LIN {X 0,Y 164.782,Z 136.258,A -85,B 0,C 180,E1 -23321.199,E2 -23321.199} C_VEL
LIN {X 0,Y 164.508,Z 136.296,A -85,B 0,C 180,E1 -23327.402,E2 -23327.402} C_VEL
LIN {X 0,Y 164.476,Z 136.307,A -85,B 0,C 180,E1 -23329.99,E2 -23329.99} C_VEL
LIN {X 0,Y 164.429,Z 136.475,A -85,B 0,C 180,E1 -23333.875,E2 -23333.875} C_VEL
LIN {X 0,Y 165.572,Z 139.373,A -85,B 0,C 180,E1 -23334.533,E2 -23334.533} C_VEL
LIN {X 0,Y 166.931,Z 141.256,A -85,B 0,C 180,E1 -23335.132,E2 -23335.132} C_VEL
LIN {X 0,Y 173.938,Z 153.479,A -85,B 0,C 180,E1 -23338.268,E2 -23338.268} C_VEL
LIN {X 0,Y 182.776,Z 169.655,A -85,B 0,C 180,E1 -23341.878,E2 -23341.878} C_VEL
LIN {X 0,Y 193.204,Z 190.491,A -85,B 0,C 180,E1 -23345.779,E2 -23345.779} C_VEL
LIN {X 0,Y 203.818,Z 212.836,A -85,B 0,C 180,E1 -23349.361,E2 -23349.361} C_VEL
LIN {X 0,Y 191.616,Z 314.791,A -85,B 0,C 180,E1 -23355.179,E2 -23355.179} C_VEL
LIN {X 0,Y 189.078,Z 333.623,A -85,B 0,C 180,E1 -23356.739,E2 -23356.739} C_VEL
LIN {X 0,Y 186.109,Z 350.938,A -85,B 0,C 180,E1 -23358.581,E2 -23358.581} C_VEL
LIN {X 0,Y 182.724,Z 368.577,A -85,B 0,C 180,E1 -23360.963,E2 -23360.963} C_VEL
LIN {X 0,Y 179.217,Z 384.609,A -85,B 0,C 180,E1 -23363.62,E2 -23363.62} C_VEL
LIN {X 0,Y 175.913,Z 399.098,A -85,B 0,C 180,E1 -23366.535,E2 -23366.535} C_VEL
LIN {X 0,Y 172.526,Z 413.606,A -85,B 0,C 180,E1 -23370.065,E2 -23370.065} C_VEL
LIN {X 0,Y 169.416,Z 427.579,A -85,B 0,C 180,E1 -23374.178,E2 -23374.178} C_VEL
LIN {X 0,Y 166.846,Z 439.432,A -85,B 0,C 180,E1 -23378.372,E2 -23378.372} C_VEL
LIN {X 0,Y 164.935,Z 449.571,A -85,B 0,C 180,E1 -23382.646,E2 -23382.646} C_VEL
LIN {X 0,Y 163.47,Z 459.455,A -85,B 0,C 180,E1 -23387.586,E2 -23387.586} C_VEL
LIN {X 0,Y 162.879,Z 465.778,A -85,B 0,C 180,E1 -23391.314,E2 -23391.314} C_VEL
LIN {X 0,Y 162.51,Z 472.942,A -85,B 0,C 180,E1 -23396.28,E2 -23396.28} C_VEL
LIN {X 0,Y 162.642,Z 478.87,A -85,B 0,C 180,E1 -23401.238,E2 -23401.238} C_VEL
LIN {X 0,Y 163.36,Z 483.627,A -85,B 0,C 180,E1 -23406.174,E2 -23406.174} C_VEL
LIN {X 0,Y 165.201,Z 488.286,A -85,B 0,C 180,E1 -23412.281,E2 -23412.281} C_VEL
LIN {X 0,Y 167.913,Z 491.025,A -85,B 0,C 180,E1 -23417.036,E2 -23417.036} C_VEL
LIN {X 0,Y 171.601,Z 493.04,A -85,B 0,C 180,E1 -23421.629,E2 -23421.629} C_VEL
LIN {X 0,Y 179.115,Z 494.623,A -85,B 0,C 180,E1 -23428.089,E2 -23428.089} C_VEL
LIN {X 0,Y 189.089,Z 494.613,A -85,B 0,C 180,E1 -23433.884,E2 -23433.884} C_VEL
LIN {X 0,Y 196.793,Z 493.837,A -85,B 0,C 180,E1 -23437.381,E2 -23437.381} C_VEL
LIN {X 0,Y 210.033,Z 491.428,A -85,B 0,C 180,E1 -23442.007,E2 -23442.007} C_VEL
LIN {X 0,Y 195.119,Z 497.326,A -85,B 0,C 180,E1 -23446.813,E2 -23446.813} C_VEL
LIN {X 0,Y 183.475,Z 501.617,A -85,B 0,C 180,E1 -23452.2,E2 -23452.2} C_VEL
LIN {X 0,Y 175.646,Z 504.236,A -85,B 0,C 180,E1 -23457.167,E2 -23457.167} C_VEL
LIN {X 0,Y 169.36,Z 505.964,A -85,B 0,C 180,E1 -23462.839,E2 -23462.839} C_VEL
LIN {X 0,Y 164.641,Z 506.692,A -85,B 0,C 180,E1 -23470.179,E2 -23470.179} C_VEL
LIN {X 0,Y 162.82,Z 505.777,A -85,B 0,C 180,E1 -23477.535,E2 -23477.535} C_VEL
LIN {X 0,Y 162.814,Z 504.732,A -85,B 0,C 180,E1 -23480.877,E2 -23480.877} C_VEL
LIN {X 0,Y 162.399,Z 503.811,A -85,B 0,C 180,E1 -23482.926,E2 -23482.926} C_VEL
LIN {X 0,Y 161.187,Z 502.51,A -85,B 0,C 180,E1 -23484.934,E2 -23484.934} C_VEL
LIN {X 0,Y 157.491,Z 497.688,A -85,B 0,C 180,E1 -23490.301,E2 -23490.301} C_VEL
LIN {X 0,Y 157.2,Z 496.337,A -85,B 0,C 180,E1 -23491.68,E2 -23491.68} C_VEL
LIN {X 0,Y 157.104,Z 492.695,A -85,B 0,C 180,E1 -23495.131,E2 -23495.131} C_VEL
LIN {X 0,Y 156.843,Z 485.87,A -85,B 0,C 180,E1 -23500.324,E2 -23500.324} C_VEL
LIN {X 0,Y 157.182,Z 479.569,A -85,B 0,C 180,E1 -23504.234,E2 -23504.234} C_VEL
LIN {X 0,Y 158.14,Z 470.979,A -85,B 0,C 180,E1 -23508.794,E2 -23508.794} C_VEL
LIN {X 0,Y 159.756,Z 460.712,A -85,B 0,C 180,E1 -23513.322,E2 -23513.322} C_VEL
LIN {X 0,Y 162.296,Z 448.632,A -85,B 0,C 180,E1 -23517.742,E2 -23517.742} C_VEL
LIN {X 0,Y 165.078,Z 436.661,A -85,B 0,C 180,E1 -23521.388,E2 -23521.388} C_VEL
LIN {X 0,Y 168.577,Z 422.487,A -85,B 0,C 180,E1 -23524.974,E2 -23524.974} C_VEL
LIN {X 0,Y 172.253,Z 407.32,A -85,B 0,C 180,E1 -23528.103,E2 -23528.103} C_VEL
LIN {X 0,Y 175.841,Z 391.722,A -85,B 0,C 180,E1 -23530.722,E2 -23530.722} C_VEL
LIN {X 0,Y 179.532,Z 374.404,A -85,B 0,C 180,E1 -23533.046,E2 -23533.046} C_VEL
LIN {X 0,Y 182.942,Z 356.554,A -85,B 0,C 180,E1 -23534.9,E2 -23534.9} C_VEL
LIN {X 0,Y 185.607,Z 338.247,A -85,B 0,C 180,E1 -23536.35,E2 -23536.35} C_VEL
LIN {X 0,Y 199.629,Z 227.884,A -85,B 0,C 180,E1 -23542.848,E2 -23542.848} C_VEL
LIN {X 0,Y 190.678,Z 205.57,A -85,B 0,C 180,E1 -23546.198,E2 -23546.198} C_VEL
LIN {X 0,Y 181.033,Z 183.19,A -85,B 0,C 180,E1 -23550.094,E2 -23550.094} C_VEL
LIN {X 0,Y 172.608,Z 164.737,A -85,B 0,C 180,E1 -23553.83,E2 -23553.83} C_VEL
LIN {X 0,Y 168.302,Z 156.399,A -85,B 0,C 180,E1 -23555.815,E2 -23555.815} C_VEL
LIN {X 0,Y 161.572,Z 145.068,A -85,B 0,C 180,E1 -23558.97,E2 -23558.97} C_VEL
LIN {X 0,Y 159.276,Z 141.104,A -85,B 0,C 180,E1 -23560.142,E2 -23560.142} C_VEL
LIN {X 0,Y 157.757,Z 138.666,A -85,B 0,C 180,E1 -23560.916,E2 -23560.916} C_VEL
LIN {X 0,Y 157.409,Z 137.193,A -85,B 0,C 180,E1 -23561.216,E2 -23561.216} C_VEL
LIN {X 0,Y 157.556,Z 137.159,A -85,B 0,C 180,E1 -23567.113,E2 -23567.113} C_VEL
LIN {X 0,Y 157.768,Z 137.14,A -85,B 0,C 180,E1 -23569.736,E2 -23569.736} C_VEL
LIN {X 0,Y 157.82,Z 137.138,A -85,B 0,C 180,E1 -23572.323,E2 -23572.323} C_VEL
LIN {X 0,Y 158.256,Z 137.083,A -85,B 0,C 180,E1 -23580,E2 -23580} C_VEL
LIN {X 0,Y 157.821,Z 137.137,A -85,B 0,C 180,E1 -23587.678,E2 -23587.678} C_VEL
LIN {X 0,Y 157.702,Z 137.147,A -85,B 0,C 180,E1 -23591.363,E2 -23591.363} C_VEL
LIN {X 0,Y 157.474,Z 137.18,A -85,B 0,C 180,E1 -23595.532,E2 -23595.532} C_VEL
LIN {X 0,Y 157.366,Z 137.196,A -85,B 0,C 180,E1 -23600.934,E2 -23600.934} C_VEL
LIN {X 0,Y 157.312,Z 137.2,A -85,B 0,C 180,E1 -23606.686,E2 -23606.686} C_VEL
LIN {X 0,Y 157.272,Z 137.2,A -85,B 0,C 180,E1 -23612.428,E2 -23612.428} C_VEL
LIN {X 0,Y 157.264,Z 137.206,A -85,B 0,C 180,E1 -23616.45,E2 -23616.45} C_VEL
LIN {X 0,Y 157.208,Z 137.214,A -85,B 0,C 180,E1 -23622.112,E2 -23622.112} C_VEL
LIN {X 0,Y 157.238,Z 137.205,A -85,B 0,C 180,E1 -23627.901,E2 -23627.901} C_VEL
LIN {X 0,Y 157.32,Z 137.189,A -85,B 0,C 180,E1 -23633.526,E2 -23633.526} C_VEL
LIN {X 0,Y 157.293,Z 137.204,A -85,B 0,C 180,E1 -23638.097,E2 -23638.097} C_VEL
LIN {X 0,Y 157.321,Z 137.198,A -85,B 0,C 180,E1 -23643.468,E2 -23643.468} C_VEL
LIN {X 0,Y 157.446,Z 137.178,A -85,B 0,C 180,E1 -23649.618,E2 -23649.618} C_VEL
LIN {X 0,Y 157.466,Z 137.175,A -85,B 0,C 180,E1 -23654.469,E2 -23654.469} C_VEL
LIN {X 0,Y 157.75,Z 137.146,A -85,B 0,C 180,E1 -23659.736,E2 -23659.736} C_VEL
LIN {X 0,Y 157.822,Z 137.133,A -85,B 0,C 180,E1 -23662.324,E2 -23662.324} C_VEL
LIN {X 0,Y 158.259,Z 137.083,A -85,B 0,C 180,E1 -23670.002,E2 -23670.002} C_VEL
LIN {X 0,Y 157.826,Z 137.141,A -85,B 0,C 180,E1 -23677.679,E2 -23677.679} C_VEL
LIN {X 0,Y 157.708,Z 137.139,A -85,B 0,C 180,E1 -23681.364,E2 -23681.364} C_VEL
LIN {X 0,Y 157.481,Z 137.184,A -85,B 0,C 180,E1 -23685.533,E2 -23685.533} C_VEL
LIN {X 0,Y 157.373,Z 137.195,A -85,B 0,C 180,E1 -23690.934,E2 -23690.934} C_VEL
LIN {X 0,Y 157.348,Z 137.194,A -85,B 0,C 180,E1 -23691.71,E2 -23691.71} C_VEL
LIN {X 0,Y 158.41,Z 140.134,A -85,B 0,C 180,E1 -23692.414,E2 -23692.414} C_VEL
LIN {X 0,Y 159.928,Z 142.172,A -85,B 0,C 180,E1 -23693.128,E2 -23693.128} C_VEL
LIN {X 0,Y 167.079,Z 154.486,A -85,B 0,C 180,E1 -23696.549,E2 -23696.549} C_VEL
LIN {X 0,Y 175.9,Z 170.567,A -85,B 0,C 180,E1 -23700.378,E2 -23700.378} C_VEL
LIN {X 0,Y 186.553,Z 191.815,A -85,B 0,C 180,E1 -23704.595,E2 -23704.595} C_VEL
LIN {X 0,Y 197.438,Z 214.94,A -85,B 0,C 180,E1 -23708.461,E2 -23708.461} C_VEL
LIN {X 0,Y 185.105,Z 314.275,A -85,B 0,C 180,E1 -23714.319,E2 -23714.319} C_VEL
LIN {X 0,Y 182.501,Z 333.276,A -85,B 0,C 180,E1 -23715.927,E2 -23715.927} C_VEL
LIN {X 0,Y 179.205,Z 352.05,A -85,B 0,C 180,E1 -23717.998,E2 -23717.998} C_VEL
LIN {X 0,Y 175.967,Z 368.444,A -85,B 0,C 180,E1 -23720.28,E2 -23720.28} C_VEL
LIN {X 0,Y 172.363,Z 384.5,A -85,B 0,C 180,E1 -23723.028,E2 -23723.028} C_VEL
LIN {X 0,Y 168.77,Z 399.805,A -85,B 0,C 180,E1 -23726.229,E2 -23726.229} C_VEL
LIN {X 0,Y 165.206,Z 414.682,A -85,B 0,C 180,E1 -23730.009,E2 -23730.009} C_VEL
LIN {X 0,Y 162.073,Z 428.527,A -85,B 0,C 180,E1 -23734.301,E2 -23734.301} C_VEL
LIN {X 0,Y 159.483,Z 440.457,A -85,B 0,C 180,E1 -23738.754,E2 -23738.754} C_VEL
LIN {X 0,Y 157.881,Z 449.027,A -85,B 0,C 180,E1 -23742.514,E2 -23742.514} C_VEL
LIN {X 0,Y 156.373,Z 459.064,A -85,B 0,C 180,E1 -23747.673,E2 -23747.673} C_VEL
LIN {X 0,Y 155.681,Z 466.451,A -85,B 0,C 180,E1 -23752.216,E2 -23752.216} C_VEL
LIN {X 0,Y 155.485,Z 473.586,A -85,B 0,C 180,E1 -23757.409,E2 -23757.409} C_VEL
LIN {X 0,Y 155.73,Z 479.475,A -85,B 0,C 180,E1 -23762.586,E2 -23762.586} C_VEL
LIN {X 0,Y 156.598,Z 484.232,A -85,B 0,C 180,E1 -23767.737,E2 -23767.737} C_VEL
LIN {X 0,Y 158.266,Z 488.082,A -85,B 0,C 180,E1 -23772.828,E2 -23772.828} C_VEL
LIN {X 0,Y 161.129,Z 491.113,A -85,B 0,C 180,E1 -23777.777,E2 -23777.777} C_VEL
LIN {X 0,Y 167.394,Z 494.193,A -85,B 0,C 180,E1 -23784.825,E2 -23784.825} C_VEL
LIN {X 0,Y 176.084,Z 495.685,A -85,B 0,C 180,E1 -23791.256,E2 -23791.256} C_VEL
LIN {X 0,Y 187.203,Z 495.638,A -85,B 0,C 180,E1 -23796.918,E2 -23796.918} C_VEL
LIN {X 0,Y 200.238,Z 494.178,A -85,B 0,C 180,E1 -23801.825,E2 -23801.825} C_VEL
LIN {X 0,Y 199.396,Z 494.527,A -85,B 0,C 180,E1 -23802.252,E2 -23802.252} C_VEL
LIN {X 0,Y 190.006,Z 497.729,A -85,B 0,C 180,E1 -23805.348,E2 -23805.348} C_VEL
LIN {X 0,Y 177.876,Z 501.623,A -85,B 0,C 180,E1 -23810.788,E2 -23810.788} C_VEL
LIN {X 0,Y 168.063,Z 504.222,A -85,B 0,C 180,E1 -23817.067,E2 -23817.067} C_VEL
LIN {X 0,Y 161.011,Z 505.535,A -85,B 0,C 180,E1 -23824.118,E2 -23824.118} C_VEL
LIN {X 0,Y 158.018,Z 505.611,A -85,B 0,C 180,E1 -23829.155,E2 -23829.155} C_VEL
LIN {X 0,Y 156.306,Z 505,A -85,B 0,C 180,E1 -23834.347,E2 -23834.347} C_VEL
LIN {X 0,Y 155.909,Z 503.121,A -85,B 0,C 180,E1 -23840.876,E2 -23840.876} C_VEL
LIN {X 0,Y 156.452,Z 501.308,A -85,B 0,C 180,E1 -23844.844,E2 -23844.844} C_VEL
LIN {X 0,Y 156.936,Z 499.805,A -85,B 0,C 180,E1 -23847.432,E2 -23847.432} C_VEL
LIN {X 0,Y 157.29,Z 497.859,A -85,B 0,C 180,E1 -23849.998,E2 -23849.998} C_VEL
LIN {X 0,Y 157.2,Z 496.337,A -85,B 0,C 180,E1 -23851.68,E2 -23851.68} C_VEL
LIN {X 0,Y 156.469,Z 494.187,A -85,B 0,C 180,E1 -23853.65,E2 -23853.65} C_VEL
LIN {X 0,Y 154.839,Z 491.662,A -85,B 0,C 180,E1 -23855.53,E2 -23855.53} C_VEL
LIN {X 0,Y 151.087,Z 485.896,A -85,B 0,C 180,E1 -23859.235,E2 -23859.235} C_VEL
LIN {X 0,Y 150.093,Z 482.788,A -85,B 0,C 180,E1 -23861.176,E2 -23861.176} C_VEL
LIN {X 0,Y 150.043,Z 481.776,A -85,B 0,C 180,E1 -23861.842,E2 -23861.842} C_VEL
LIN {X 0,Y 150.725,Z 473.135,A -85,B 0,C 180,E1 -23866.941,E2 -23866.941} C_VEL
LIN {X 0,Y 152.057,Z 463.428,A -85,B 0,C 180,E1 -23871.699,E2 -23871.699} C_VEL
LIN {X 0,Y 154.322,Z 452.034,A -85,B 0,C 180,E1 -23876.359,E2 -23876.359} C_VEL
LIN {X 0,Y 157.22,Z 439.664,A -85,B 0,C 180,E1 -23880.561,E2 -23880.561} C_VEL
LIN {X 0,Y 160.831,Z 425.013,A -85,B 0,C 180,E1 -23884.614,E2 -23884.614} C_VEL
LIN {X 0,Y 164.79,Z 408.962,A -85,B 0,C 180,E1 -23888.197,E2 -23888.197} C_VEL
LIN {X 0,Y 168.826,Z 392.119,A -85,B 0,C 180,E1 -23891.203,E2 -23891.203} C_VEL
LIN {X 0,Y 172.548,Z 375.19,A -85,B 0,C 180,E1 -23893.598,E2 -23893.598} C_VEL
LIN {X 0,Y 176.029,Z 357.565,A -85,B 0,C 180,E1 -23895.532,E2 -23895.532} C_VEL
LIN {X 0,Y 178.683,Z 340.392,A -85,B 0,C 180,E1 -23896.996,E2 -23896.996} C_VEL
LIN {X 0,Y 193.251,Z 229.764,A -85,B 0,C 180,E1 -23903.774,E2 -23903.774} C_VEL
LIN {X 0,Y 185.238,Z 209.471,A -85,B 0,C 180,E1 -23906.908,E2 -23906.908} C_VEL
LIN {X 0,Y 175.951,Z 187.639,A -85,B 0,C 180,E1 -23910.826,E2 -23910.826} C_VEL
LIN {X 0,Y 167.779,Z 169.366,A -85,B 0,C 180,E1 -23914.625,E2 -23914.625} C_VEL
LIN {X 0,Y 163.269,Z 160.612,A -85,B 0,C 180,E1 -23916.777,E2 -23916.777} C_VEL
LIN {X 0,Y 156.306,Z 148.806,A -85,B 0,C 180,E1 -23920.21,E2 -23920.21} C_VEL
LIN {X 0,Y 154.262,Z 145.429,A -85,B 0,C 180,E1 -23921.286,E2 -23921.286} C_VEL
LIN {X 0,Y 152.425,Z 142.211,A -85,B 0,C 180,E1 -23922.301,E2 -23922.301} C_VEL
LIN {X 0,Y 150.837,Z 139.865,A -85,B 0,C 180,E1 -23923.157,E2 -23923.157} C_VEL
LIN {X 0,Y 150.378,Z 138.061,A -85,B 0,C 180,E1 -23923.628,E2 -23923.628} C_VEL
LIN {X 0,Y 150.685,Z 138.018,A -85,B 0,C 180,E1 -23929.248,E2 -23929.248} C_VEL
LIN {X 0,Y 150.759,Z 138.019,A -85,B 0,C 180,E1 -23931.961,E2 -23931.961} C_VEL
LIN {X 0,Y 151.216,Z 137.96,A -85,B 0,C 180,E1 -23940,E2 -23940} C_VEL
LIN {X 0,Y 150.759,Z 138.019,A -85,B 0,C 180,E1 -23948.04,E2 -23948.04} C_VEL
LIN {X 0,Y 150.631,Z 138.027,A -85,B 0,C 180,E1 -23951.546,E2 -23951.546} C_VEL
LIN {X 0,Y 150.379,Z 138.061,A -85,B 0,C 180,E1 -23956.285,E2 -23956.285} C_VEL
LIN {X 0,Y 150.347,Z 138.07,A -85,B 0,C 180,E1 -23960.793,E2 -23960.793} C_VEL
LIN {X 0,Y 150.241,Z 138.084,A -85,B 0,C 180,E1 -23967.283,E2 -23967.283} C_VEL
LIN {X 0,Y 150.212,Z 138.08,A -85,B 0,C 180,E1 -23972.634,E2 -23972.634} C_VEL
LIN {X 0,Y 150.169,Z 138.083,A -85,B 0,C 180,E1 -23977.475,E2 -23977.475} C_VEL
LIN {X 0,Y 150.148,Z 138.094,A -85,B 0,C 180,E1 -23981.506,E2 -23981.506} C_VEL
LIN {X 0,Y 150.14,Z 138.085,A -85,B 0,C 180,E1 -23985.403,E2 -23985.403} C_VEL
LIN {X 0,Y 150.186,Z 138.087,A -85,B 0,C 180,E1 -23989.073,E2 -23989.073} C_VEL
LIN {X 0,Y 150.228,Z 138.076,A -85,B 0,C 180,E1 -23992.684,E2 -23992.684} C_VEL
LIN {X 0,Y 150.217,Z 138.085,A -85,B 0,C 180,E1 -23997.367,E2 -23997.367} C_VEL
LIN {X 0,Y 150.243,Z 138.073,A -85,B 0,C 180,E1 -24002.72,E2 -24002.72} C_VEL
LIN {X 0,Y 150.389,Z 138.055,A -85,B 0,C 180,E1 -24009.171,E2 -24009.171} C_VEL
LIN {X 0,Y 150.377,Z 138.063,A -85,B 0,C 180,E1 -24013.717,E2 -24013.717} C_VEL
LIN {X 0,Y 150.664,Z 138.03,A -85,B 0,C 180,E1 -24019.248,E2 -24019.248} C_VEL
LIN {X 0,Y 150.757,Z 138.011,A -85,B 0,C 180,E1 -24021.962,E2 -24021.962} C_VEL
LIN {X 0,Y 151.22,Z 137.96,A -85,B 0,C 180,E1 -24030.002,E2 -24030.002} C_VEL
LIN {X 0,Y 150.765,Z 138.022,A -85,B 0,C 180,E1 -24038.041,E2 -24038.041} C_VEL
LIN {X 0,Y 150.637,Z 138.019,A -85,B 0,C 180,E1 -24041.547,E2 -24041.547} C_VEL
LIN {X 0,Y 150.385,Z 138.063,A -85,B 0,C 180,E1 -24046.286,E2 -24046.286} C_VEL
LIN {X 0,Y 150.355,Z 138.174,A -85,B 0,C 180,E1 -24049.439,E2 -24049.439} C_VEL
LIN {X 0,Y 151.372,Z 140.924,A -85,B 0,C 180,E1 -24050.145,E2 -24050.145} C_VEL
LIN {X 0,Y 153.026,Z 143.281,A -85,B 0,C 180,E1 -24051.003,E2 -24051.003} C_VEL
LIN {X 0,Y 161.514,Z 157.586,A -85,B 0,C 180,E1 -24055.299,E2 -24055.299} C_VEL
LIN {X 0,Y 170.853,Z 174.947,A -85,B 0,C 180,E1 -24059.58,E2 -24059.58} C_VEL
LIN {X 0,Y 181.271,Z 195.919,A -85,B 0,C 180,E1 -24063.873,E2 -24063.873} C_VEL
LIN {X 0,Y 191.032,Z 216.93,A -85,B 0,C 180,E1 -24067.503,E2 -24067.503} C_VEL
LIN {X 0,Y 178.361,Z 316.308,A -85,B 0,C 180,E1 -24073.611,E2 -24073.611} C_VEL
LIN {X 0,Y 175.544,Z 335.304,A -85,B 0,C 180,E1 -24075.322,E2 -24075.322} C_VEL
LIN {X 0,Y 172.298,Z 353.063,A -85,B 0,C 180,E1 -24077.383,E2 -24077.383} C_VEL
LIN {X 0,Y 168.884,Z 369.821,A -85,B 0,C 180,E1 -24079.832,E2 -24079.832} C_VEL
LIN {X 0,Y 164.874,Z 387.158,A -85,B 0,C 180,E1 -24082.98,E2 -24082.98} C_VEL
LIN {X 0,Y 161.038,Z 403.06,A -85,B 0,C 180,E1 -24086.566,E2 -24086.566} C_VEL
LIN {X 0,Y 157.418,Z 417.671,A -85,B 0,C 180,E1 -24090.587,E2 -24090.587} C_VEL
LIN {X 0,Y 154.771,Z 429.392,A -85,B 0,C 180,E1 -24094.444,E2 -24094.444} C_VEL
LIN {X 0,Y 151.912,Z 442.604,A -85,B 0,C 180,E1 -24099.697,E2 -24099.697} C_VEL
LIN {X 0,Y 150.136,Z 452.395,A -85,B 0,C 180,E1 -24104.385,E2 -24104.385} C_VEL
LIN {X 0,Y 149.062,Z 460.821,A -85,B 0,C 180,E1 -24109.129,E2 -24109.129} C_VEL
LIN {X 0,Y 148.494,Z 467.747,A -85,B 0,C 180,E1 -24113.682,E2 -24113.682} C_VEL
LIN {X 0,Y 148.431,Z 474.157,A -85,B 0,C 180,E1 -24118.643,E2 -24118.643} C_VEL
LIN {X 0,Y 148.856,Z 480.016,A -85,B 0,C 180,E1 -24124.061,E2 -24124.061} C_VEL
LIN {X 0,Y 149.874,Z 484.762,A -85,B 0,C 180,E1 -24129.415,E2 -24129.415} C_VEL
LIN {X 0,Y 152.761,Z 489.541,A -85,B 0,C 180,E1 -24136.024,E2 -24136.024} C_VEL
LIN {X 0,Y 158.482,Z 493.563,A -85,B 0,C 180,E1 -24143.522,E2 -24143.522} C_VEL
LIN {X 0,Y 166.753,Z 495.963,A -85,B 0,C 180,E1 -24150.381,E2 -24150.381} C_VEL
LIN {X 0,Y 177.61,Z 496.835,A -85,B 0,C 180,E1 -24156.409,E2 -24156.409} C_VEL
LIN {X 0,Y 185.932,Z 496.689,A -85,B 0,C 180,E1 -24159.984,E2 -24159.984} C_VEL
LIN {X 0,Y 190.453,Z 496.319,A -85,B 0,C 180,E1 -24161.623,E2 -24161.623} C_VEL
LIN {X 0,Y 189.726,Z 496.644,A -85,B 0,C 180,E1 -24162.193,E2 -24162.193} C_VEL
LIN {X 0,Y 176.334,Z 500.455,A -85,B 0,C 180,E1 -24167.345,E2 -24167.345} C_VEL
LIN {X 0,Y 165.199,Z 503.044,A -85,B 0,C 180,E1 -24173.443,E2 -24173.443} C_VEL
LIN {X 0,Y 156.735,Z 504.437,A -85,B 0,C 180,E1 -24180.444,E2 -24180.444} C_VEL
LIN {X 0,Y 151.318,Z 504.497,A -85,B 0,C 180,E1 -24188.263,E2 -24188.263} C_VEL
LIN {X 0,Y 149.085,Z 502.965,A -85,B 0,C 180,E1 -24196.365,E2 -24196.365} C_VEL
LIN {X 0,Y 149.154,Z 500.975,A -85,B 0,C 180,E1 -24201.872,E2 -24201.872} C_VEL
LIN {X 0,Y 150.088,Z 497.95,A -85,B 0,C 180,E1 -24207.314,E2 -24207.314} C_VEL
LIN {X 0,Y 150.426,Z 495.968,A -85,B 0,C 180,E1 -24209.998,E2 -24209.998} C_VEL
LIN {X 0,Y 150.285,Z 492.026,A -85,B 0,C 180,E1 -24214.021,E2 -24214.021} C_VEL
LIN {X 0,Y 149.972,Z 487.115,A -85,B 0,C 180,E1 -24218.08,E2 -24218.08} C_VEL
LIN {X 0,Y 150.043,Z 481.776,A -85,B 0,C 180,E1 -24221.842,E2 -24221.842} C_VEL
LIN {X 0,Y 149.544,Z 478.645,A -85,B 0,C 180,E1 -24223.748,E2 -24223.748} C_VEL
LIN {X 0,Y 147.183,Z 472.836,A -85,B 0,C 180,E1 -24226.72,E2 -24226.72} C_VEL
LIN {X 0,Y 145.065,Z 466.576,A -85,B 0,C 180,E1 -24229.66,E2 -24229.66} C_VEL
LIN {X 0,Y 144.996,Z 462.716,A -85,B 0,C 180,E1 -24231.455,E2 -24231.455} C_VEL
LIN {X 0,Y 147.162,Z 451.704,A -85,B 0,C 180,E1 -24236.214,E2 -24236.214} C_VEL
LIN {X 0,Y 150.056,Z 439.396,A -85,B 0,C 180,E1 -24240.618,E2 -24240.618} C_VEL
LIN {X 0,Y 153.576,Z 425.04,A -85,B 0,C 180,E1 -24244.819,E2 -24244.819} C_VEL
LIN {X 0,Y 157.351,Z 410.447,A -85,B 0,C 180,E1 -24248.293,E2 -24248.293} C_VEL
LIN {X 0,Y 161.514,Z 393.739,A -85,B 0,C 180,E1 -24251.49,E2 -24251.49} C_VEL
LIN {X 0,Y 165.299,Z 377.248,A -85,B 0,C 180,E1 -24253.994,E2 -24253.994} C_VEL
LIN {X 0,Y 168.868,Z 359.619,A -85,B 0,C 180,E1 -24256.095,E2 -24256.095} C_VEL
LIN {X 0,Y 171.879,Z 341.858,A -85,B 0,C 180,E1 -24257.715,E2 -24257.715} C_VEL
LIN {X 0,Y 186.866,Z 231.166,A -85,B 0,C 180,E1 -24264.786,E2 -24264.786} C_VEL
LIN {X 0,Y 176.346,Z 204.988,A -85,B 0,C 180,E1 -24269.129,E2 -24269.129} C_VEL
LIN {X 0,Y 166.945,Z 183.018,A -85,B 0,C 180,E1 -24273.447,E2 -24273.447} C_VEL
LIN {X 0,Y 160.223,Z 168.344,A -85,B 0,C 180,E1 -24276.813,E2 -24276.813} C_VEL
LIN {X 0,Y 152.52,Z 154.871,A -85,B 0,C 180,E1 -24280.747,E2 -24280.747} C_VEL
LIN {X 0,Y 147.962,Z 147.258,A -85,B 0,C 180,E1 -24283.264,E2 -24283.264} C_VEL
LIN {X 0,Y 146.03,Z 143.895,A -85,B 0,C 180,E1 -24284.419,E2 -24284.419} C_VEL
LIN {X 0,Y 143.958,Z 140.994,A -85,B 0,C 180,E1 -24285.601,E2 -24285.601} C_VEL
LIN {X 0,Y 143.396,Z 138.928,A -85,B 0,C 180,E1 -24286.177,E2 -24286.177} C_VEL
LIN {X 0,Y 143.596,Z 138.897,A -85,B 0,C 180,E1 -24288.711,E2 -24288.711} C_VEL
LIN {X 0,Y 143.681,Z 138.903,A -85,B 0,C 180,E1 -24291.562,E2 -24291.562} C_VEL
LIN {X 0,Y 144.175,Z 138.837,A -85,B 0,C 180,E1 -24300,E2 -24300} C_VEL
LIN {X 0,Y 143.681,Z 138.9,A -85,B 0,C 180,E1 -24308.438,E2 -24308.438} C_VEL
LIN {X 0,Y 143.567,Z 138.906,A -85,B 0,C 180,E1 -24311.758,E2 -24311.758} C_VEL
LIN {X 0,Y 143.313,Z 138.937,A -85,B 0,C 180,E1 -24317.112,E2 -24317.112} C_VEL
LIN {X 0,Y 143.273,Z 138.951,A -85,B 0,C 180,E1 -24321.256,E2 -24321.256} C_VEL
LIN {X 0,Y 143.187,Z 138.961,A -85,B 0,C 180,E1 -24327.939,E2 -24327.939} C_VEL
LIN {X 0,Y 143.161,Z 138.962,A -85,B 0,C 180,E1 -24333.434,E2 -24333.434} C_VEL
LIN {X 0,Y 143.058,Z 138.967,A -85,B 0,C 180,E1 -24339.691,E2 -24339.691} C_VEL
LIN {X 0,Y 143.059,Z 138.975,A -85,B 0,C 180,E1 -24343.454,E2 -24343.454} C_VEL
LIN {X 0,Y 143.086,Z 138.963,A -85,B 0,C 180,E1 -24347.456,E2 -24347.456} C_VEL
LIN {X 0,Y 143.123,Z 138.966,A -85,B 0,C 180,E1 -24351.783,E2 -24351.783} C_VEL
LIN {X 0,Y 143.184,Z 138.961,A -85,B 0,C 180,E1 -24357.324,E2 -24357.324} C_VEL
LIN {X 0,Y 143.162,Z 138.962,A -85,B 0,C 180,E1 -24363.782,E2 -24363.782} C_VEL
LIN {X 0,Y 143.34,Z 138.936,A -85,B 0,C 180,E1 -24369.929,E2 -24369.929} C_VEL
LIN {X 0,Y 143.372,Z 138.929,A -85,B 0,C 180,E1 -24375.814,E2 -24375.814} C_VEL
LIN {X 0,Y 143.595,Z 138.911,A -85,B 0,C 180,E1 -24378.712,E2 -24378.712} C_VEL
LIN {X 0,Y 143.676,Z 138.892,A -85,B 0,C 180,E1 -24381.563,E2 -24381.563} C_VEL
LIN {X 0,Y 144.178,Z 138.837,A -85,B 0,C 180,E1 -24390.002,E2 -24390.002} C_VEL
LIN {X 0,Y 143.687,Z 138.902,A -85,B 0,C 180,E1 -24398.44,E2 -24398.44} C_VEL
LIN {X 0,Y 143.574,Z 138.898,A -85,B 0,C 180,E1 -24401.76,E2 -24401.76} C_VEL
LIN {X 0,Y 143.318,Z 138.937,A -85,B 0,C 180,E1 -24406.838,E2 -24406.838} C_VEL
LIN {X 0,Y 144.282,Z 141.767,A -85,B 0,C 180,E1 -24407.635,E2 -24407.635} C_VEL
LIN {X 0,Y 146.024,Z 144.042,A -85,B 0,C 180,E1 -24408.596,E2 -24408.596} C_VEL
LIN {X 0,Y 153.528,Z 156.749,A -85,B 0,C 180,E1 -24412.767,E2 -24412.767} C_VEL
LIN {X 0,Y 159.504,Z 167.387,A -85,B 0,C 180,E1 -24415.784,E2 -24415.784} C_VEL
LIN {X 0,Y 167.995,Z 183.583,A -85,B 0,C 180,E1 -24419.725,E2 -24419.725} C_VEL
LIN {X 0,Y 177.519,Z 203.382,A -85,B 0,C 180,E1 -24423.758,E2 -24423.758} C_VEL
LIN {X 0,Y 184.701,Z 218.997,A -85,B 0,C 180,E1 -24426.525,E2 -24426.525} C_VEL
LIN {X 0,Y 171.836,Z 316.112,A -85,B 0,C 180,E1 -24432.7,E2 -24432.7} C_VEL
LIN {X 0,Y 168.823,Z 335.86,A -85,B 0,C 180,E1 -24434.528,E2 -24434.528} C_VEL
LIN {X 0,Y 165.463,Z 353.711,A -85,B 0,C 180,E1 -24436.688,E2 -24436.688} C_VEL
LIN {X 0,Y 161.794,Z 371.023,A -85,B 0,C 180,E1 -24439.34,E2 -24439.34} C_VEL
LIN {X 0,Y 158.061,Z 386.784,A -85,B 0,C 180,E1 -24442.311,E2 -24442.311} C_VEL
LIN {X 0,Y 154.323,Z 401.9,A -85,B 0,C 180,E1 -24445.799,E2 -24445.799} C_VEL
LIN {X 0,Y 150.622,Z 416.431,A -85,B 0,C 180,E1 -24449.894,E2 -24449.894} C_VEL
LIN {X 0,Y 147.883,Z 428.286,A -85,B 0,C 180,E1 -24453.922,E2 -24453.922} C_VEL
LIN {X 0,Y 145.201,Z 440.142,A -85,B 0,C 180,E1 -24458.714,E2 -24458.714} C_VEL
LIN {X 0,Y 143.29,Z 450.366,A -85,B 0,C 180,E1 -24463.619,E2 -24463.619} C_VEL
LIN {X 0,Y 141.979,Z 460.294,A -85,B 0,C 180,E1 -24469.302,E2 -24469.302} C_VEL
LIN {X 0,Y 141.442,Z 467.599,A -85,B 0,C 180,E1 -24474.296,E2 -24474.296} C_VEL
LIN {X 0,Y 141.43,Z 474.664,A -85,B 0,C 180,E1 -24480,E2 -24480} C_VEL
LIN {X 0,Y 142.073,Z 480.497,A -85,B 0,C 180,E1 -24485.678,E2 -24485.678} C_VEL
LIN {X 0,Y 143.881,Z 486.322,A -85,B 0,C 180,E1 -24492.697,E2 -24492.697} C_VEL
LIN {X 0,Y 147.656,Z 490.871,A -85,B 0,C 180,E1 -24499.462,E2 -24499.462} C_VEL
LIN {X 0,Y 154.628,Z 494.738,A -85,B 0,C 180,E1 -24507.033,E2 -24507.033} C_VEL
LIN {X 0,Y 164.156,Z 497.073,A -85,B 0,C 180,E1 -24513.818,E2 -24513.818} C_VEL
LIN {X 0,Y 176.196,Z 497.914,A -85,B 0,C 180,E1 -24519.657,E2 -24519.657} C_VEL
LIN {X 0,Y 180.625,Z 497.88,A -85,B 0,C 180,E1 -24521.411,E2 -24521.411} C_VEL
LIN {X 0,Y 180.159,Z 498.183,A -85,B 0,C 180,E1 -24522.165,E2 -24522.165} C_VEL
LIN {X 0,Y 167.041,Z 501.171,A -85,B 0,C 180,E1 -24527.685,E2 -24527.685} C_VEL
LIN {X 0,Y 156.208,Z 502.977,A -85,B 0,C 180,E1 -24534.203,E2 -24534.203} C_VEL
LIN {X 0,Y 148.277,Z 503.559,A -85,B 0,C 180,E1 -24541.705,E2 -24541.705} C_VEL
LIN {X 0,Y 143.559,Z 502.808,A -85,B 0,C 180,E1 -24549.957,E2 -24549.957} C_VEL
LIN {X 0,Y 142.107,Z 500.434,A -85,B 0,C 180,E1 -24558.588,E2 -24558.588} C_VEL
LIN {X 0,Y 142.684,Z 497.785,A -85,B 0,C 180,E1 -24564.345,E2 -24564.345} C_VEL
LIN {X 0,Y 143.246,Z 496.066,A -85,B 0,C 180,E1 -24567.186,E2 -24567.186} C_VEL
LIN {X 0,Y 143.574,Z 493.913,A -85,B 0,C 180,E1 -24569.998,E2 -24569.998} C_VEL
LIN {X 0,Y 143.391,Z 489.804,A -85,B 0,C 180,E1 -24574.214,E2 -24574.214} C_VEL
LIN {X 0,Y 143.06,Z 482.986,A -85,B 0,C 180,E1 -24579.689,E2 -24579.689} C_VEL
LIN {X 0,Y 143.452,Z 475.118,A -85,B 0,C 180,E1 -24584.902,E2 -24584.902} C_VEL
LIN {X 0,Y 144.507,Z 465.936,A -85,B 0,C 180,E1 -24589.902,E2 -24589.902} C_VEL
LIN {X 0,Y 144.996,Z 462.716,A -85,B 0,C 180,E1 -24591.455,E2 -24591.455} C_VEL
LIN {X 0,Y 145.029,Z 458.87,A -85,B 0,C 180,E1 -24593.189,E2 -24593.189} C_VEL
LIN {X 0,Y 143.526,Z 451.971,A -85,B 0,C 180,E1 -24595.944,E2 -24595.944} C_VEL
LIN {X 0,Y 142.214,Z 444.72,A -85,B 0,C 180,E1 -24598.649,E2 -24598.649} C_VEL
LIN {X 0,Y 142.585,Z 440.233,A -85,B 0,C 180,E1 -24600.249,E2 -24600.249} C_VEL
LIN {X 0,Y 145.932,Z 426.929,A -85,B 0,C 180,E1 -24604.461,E2 -24604.461} C_VEL
LIN {X 0,Y 149.578,Z 413.015,A -85,B 0,C 180,E1 -24608.072,E2 -24608.072} C_VEL
LIN {X 0,Y 153.807,Z 396.658,A -85,B 0,C 180,E1 -24611.493,E2 -24611.493} C_VEL
LIN {X 0,Y 157.959,Z 379.193,A -85,B 0,C 180,E1 -24614.386,E2 -24614.386} C_VEL
LIN {X 0,Y 161.78,Z 361.316,A -85,B 0,C 180,E1 -24616.687,E2 -24616.687} C_VEL
LIN {X 0,Y 164.999,Z 343.595,A -85,B 0,C 180,E1 -24618.42,E2 -24618.42} C_VEL
LIN {X 0,Y 170.674,Z 301.218,A -85,B 0,C 180,E1 -24621.476,E2 -24621.476} C_VEL
LIN {X 0,Y 180.448,Z 232.77,A -85,B 0,C 180,E1 -24625.826,E2 -24625.826} C_VEL
LIN {X 0,Y 170.594,Z 208.052,A -85,B 0,C 180,E1 -24630.107,E2 -24630.107} C_VEL
LIN {X 0,Y 161.656,Z 186.898,A -85,B 0,C 180,E1 -24634.412,E2 -24634.412} C_VEL
LIN {X 0,Y 155.164,Z 172.49,A -85,B 0,C 180,E1 -24637.827,E2 -24637.827} C_VEL
LIN {X 0,Y 147.35,Z 158.648,A -85,B 0,C 180,E1 -24642.041,E2 -24642.041} C_VEL
LIN {X 0,Y 143.031,Z 151.5,A -85,B 0,C 180,E1 -24644.556,E2 -24644.556} C_VEL
LIN {X 0,Y 140.945,Z 148.068,A -85,B 0,C 180,E1 -24645.84,E2 -24645.84} C_VEL
LIN {X 0,Y 139.126,Z 144.852,A -85,B 0,C 180,E1 -24647.047,E2 -24647.047} C_VEL
LIN {X 0,Y 137.008,Z 141.55,A -85,B 0,C 180,E1 -24648.421,E2 -24648.421} C_VEL
LIN {X 0,Y 136.569,Z 139.772,A -85,B 0,C 180,E1 -24648.948,E2 -24648.948} C_VEL
LIN {X 0,Y 136.566,Z 139.767,A -85,B 0,C 180,E1 -24654.093,E2 -24654.093} C_VEL
LIN {X 0,Y 137.132,Z 139.715,A -85,B 0,C 180,E1 -24660,E2 -24660} C_VEL
LIN {X 0,Y 136.605,Z 139.782,A -85,B 0,C 180,E1 -24668.879,E2 -24668.879} C_VEL
LIN {X 0,Y 136.489,Z 139.788,A -85,B 0,C 180,E1 -24671.958,E2 -24671.958} C_VEL
LIN {X 0,Y 136.248,Z 139.817,A -85,B 0,C 180,E1 -24678.029,E2 -24678.029} C_VEL
LIN {X 0,Y 136.195,Z 139.83,A -85,B 0,C 180,E1 -24681.75,E2 -24681.75} C_VEL
LIN {X 0,Y 136.113,Z 139.841,A -85,B 0,C 180,E1 -24688.63,E2 -24688.63} C_VEL
LIN {X 0,Y 136.068,Z 139.848,A -85,B 0,C 180,E1 -24694.622,E2 -24694.622} C_VEL
LIN {X 0,Y 136.028,Z 139.841,A -85,B 0,C 180,E1 -24699.2,E2 -24699.2} C_VEL
LIN {X 0,Y 136.001,Z 139.854,A -85,B 0,C 180,E1 -24703.662,E2 -24703.662} C_VEL
LIN {X 0,Y 136.048,Z 139.842,A -85,B 0,C 180,E1 -24707.815,E2 -24707.815} C_VEL
LIN {X 0,Y 136.073,Z 139.844,A -85,B 0,C 180,E1 -24711.702,E2 -24711.702} C_VEL
LIN {X 0,Y 136.09,Z 139.839,A -85,B 0,C 180,E1 -24715.719,E2 -24715.719} C_VEL
LIN {X 0,Y 136.146,Z 139.826,A -85,B 0,C 180,E1 -24722.319,E2 -24722.319} C_VEL
LIN {X 0,Y 136.277,Z 139.811,A -85,B 0,C 180,E1 -24728.841,E2 -24728.841} C_VEL
LIN {X 0,Y 136.281,Z 139.811,A -85,B 0,C 180,E1 -24735.06,E2 -24735.06} C_VEL
LIN {X 0,Y 136.497,Z 139.795,A -85,B 0,C 180,E1 -24738.117,E2 -24738.117} C_VEL
LIN {X 0,Y 136.6,Z 139.773,A -85,B 0,C 180,E1 -24741.123,E2 -24741.123} C_VEL
LIN {X 0,Y 137.136,Z 139.714,A -85,B 0,C 180,E1 -24750.002,E2 -24750.002} C_VEL
LIN {X 0,Y 136.611,Z 139.782,A -85,B 0,C 180,E1 -24758.88,E2 -24758.88} C_VEL
LIN {X 0,Y 136.368,Z 139.844,A -85,B 0,C 180,E1 -24764.076,E2 -24764.076} C_VEL
LIN {X 0,Y 137.222,Z 142.48,A -85,B 0,C 180,E1 -24764.84,E2 -24764.84} C_VEL
LIN {X 0,Y 139.138,Z 145.106,A -85,B 0,C 180,E1 -24766.022,E2 -24766.022} C_VEL
LIN {X 0,Y 141.271,Z 148.545,A -85,B 0,C 180,E1 -24767.369,E2 -24767.369} C_VEL
LIN {X 0,Y 148.822,Z 161.376,A -85,B 0,C 180,E1 -24771.785,E2 -24771.785} C_VEL
LIN {X 0,Y 155.664,Z 173.749,A -85,B 0,C 180,E1 -24775.382,E2 -24775.382} C_VEL
LIN {X 0,Y 164.117,Z 190.455,A -85,B 0,C 180,E1 -24779.46,E2 -24779.46} C_VEL
LIN {X 0,Y 172.873,Z 209.01,A -85,B 0,C 180,E1 -24783.289,E2 -24783.289} C_VEL
LIN {X 0,Y 178.334,Z 220.873,A -85,B 0,C 180,E1 -24785.477,E2 -24785.477} C_VEL
LIN {X 0,Y 165.25,Z 316.476,A -85,B 0,C 180,E1 -24791.79,E2 -24791.79} C_VEL
LIN {X 0,Y 162.188,Z 335.926,A -85,B 0,C 180,E1 -24793.653,E2 -24793.653} C_VEL
LIN {X 0,Y 158.608,Z 354.377,A -85,B 0,C 180,E1 -24795.963,E2 -24795.963} C_VEL
LIN {X 0,Y 155.112,Z 370.414,A -85,B 0,C 180,E1 -24798.498,E2 -24798.498} C_VEL
LIN {X 0,Y 150.904,Z 387.679,A -85,B 0,C 180,E1 -24801.896,E2 -24801.896} C_VEL
LIN {X 0,Y 146.875,Z 403.596,A -85,B 0,C 180,E1 -24805.789,E2 -24805.789} C_VEL
LIN {X 0,Y 143.35,Z 417.156,A -85,B 0,C 180,E1 -24809.833,E2 -24809.833} C_VEL
LIN {X 0,Y 140.692,Z 428.381,A -85,B 0,C 180,E1 -24813.848,E2 -24813.848} C_VEL
LIN {X 0,Y 138.229,Z 439.175,A -85,B 0,C 180,E1 -24818.37,E2 -24818.37} C_VEL
LIN {X 0,Y 136.239,Z 449.58,A -85,B 0,C 180,E1 -24823.517,E2 -24823.517} C_VEL
LIN {X 0,Y 135.062,Z 458.47,A -85,B 0,C 180,E1 -24828.747,E2 -24828.747} C_VEL
LIN {X 0,Y 134.45,Z 466.122,A -85,B 0,C 180,E1 -24833.999,E2 -24833.999} C_VEL
LIN {X 0,Y 134.425,Z 473.465,A -85,B 0,C 180,E1 -24840,E2 -24840} C_VEL
LIN {X 0,Y 135.078,Z 479.556,A -85,B 0,C 180,E1 -24845.973,E2 -24845.973} C_VEL
LIN {X 0,Y 136.995,Z 485.752,A -85,B 0,C 180,E1 -24853.347,E2 -24853.347} C_VEL
LIN {X 0,Y 140.991,Z 490.552,A -85,B 0,C 180,E1 -24860.422,E2 -24860.422} C_VEL
LIN {X 0,Y 145.577,Z 493.6,A -85,B 0,C 180,E1 -24865.753,E2 -24865.753} C_VEL
LIN {X 0,Y 154.671,Z 496.805,A -85,B 0,C 180,E1 -24873.042,E2 -24873.042} C_VEL
LIN {X 0,Y 166.477,Z 498.551,A -85,B 0,C 180,E1 -24879.289,E2 -24879.289} C_VEL
LIN {X 0,Y 171.525,Z 498.87,A -85,B 0,C 180,E1 -24881.439,E2 -24881.439} C_VEL
LIN {X 0,Y 170.692,Z 499.166,A -85,B 0,C 180,E1 -24882.17,E2 -24882.17} C_VEL
LIN {X 0,Y 157.76,Z 501.351,A -85,B 0,C 180,E1 -24888.067,E2 -24888.067} C_VEL
LIN {X 0,Y 147.348,Z 502.404,A -85,B 0,C 180,E1 -24895.083,E2 -24895.083} C_VEL
LIN {X 0,Y 139.969,Z 502.189,A -85,B 0,C 180,E1 -24903.132,E2 -24903.132} C_VEL
LIN {X 0,Y 136.943,Z 501.3,A -85,B 0,C 180,E1 -24908.944,E2 -24908.944} C_VEL
LIN {X 0,Y 135.478,Z 499.732,A -85,B 0,C 180,E1 -24914.965,E2 -24914.965} C_VEL
LIN {X 0,Y 135.439,Z 497.407,A -85,B 0,C 180,E1 -24921.042,E2 -24921.042} C_VEL
LIN {X 0,Y 136.453,Z 494.046,A -85,B 0,C 180,E1 -24927.046,E2 -24927.046} C_VEL
LIN {X 0,Y 136.746,Z 491.824,A -85,B 0,C 180,E1 -24929.998,E2 -24929.998} C_VEL
LIN {X 0,Y 136.496,Z 487.446,A -85,B 0,C 180,E1 -24934.428,E2 -24934.428} C_VEL
LIN {X 0,Y 136.242,Z 480.093,A -85,B 0,C 180,E1 -24940.377,E2 -24940.377} C_VEL
LIN {X 0,Y 136.66,Z 472.026,A -85,B 0,C 180,E1 -24945.662,E2 -24945.662} C_VEL
LIN {X 0,Y 137.848,Z 462.487,A -85,B 0,C 180,E1 -24950.907,E2 -24950.907} C_VEL
LIN {X 0,Y 139.898,Z 451.829,A -85,B 0,C 180,E1 -24955.821,E2 -24955.821} C_VEL
LIN {X 0,Y 142.585,Z 440.233,A -85,B 0,C 180,E1 -24960.249,E2 -24960.249} C_VEL
LIN {X 0,Y 143.023,Z 435.764,A -85,B 0,C 180,E1 -24961.787,E2 -24961.787} C_VEL
LIN {X 0,Y 142.141,Z 428.029,A -85,B 0,C 180,E1 -24964.25,E2 -24964.25} C_VEL
LIN {X 0,Y 141.349,Z 419.996,A -85,B 0,C 180,E1 -24966.6,E2 -24966.6} C_VEL
LIN {X 0,Y 141.929,Z 415.056,A -85,B 0,C 180,E1 -24967.908,E2 -24967.908} C_VEL
LIN {X 0,Y 146.003,Z 399.658,A -85,B 0,C 180,E1 -24971.44,E2 -24971.44} C_VEL
LIN {X 0,Y 149.807,Z 384.495,A -85,B 0,C 180,E1 -24974.251,E2 -24974.251} C_VEL
LIN {X 0,Y 153.579,Z 368.172,A -85,B 0,C 180,E1 -24976.653,E2 -24976.653} C_VEL
LIN {X 0,Y 157.259,Z 350.058,A -85,B 0,C 180,E1 -24978.706,E2 -24978.706} C_VEL
LIN {X 0,Y 160.247,Z 330.547,A -85,B 0,C 180,E1 -24980.373,E2 -24980.373} C_VEL
LIN {X 0,Y 174.075,Z 234.51,A -85,B 0,C 180,E1 -24986.892,E2 -24986.892} C_VEL
LIN {X 0,Y 164.532,Z 210.269,A -85,B 0,C 180,E1 -24991.279,E2 -24991.279} C_VEL
LIN {X 0,Y 155.776,Z 189.313,A -85,B 0,C 180,E1 -24995.762,E2 -24995.762} C_VEL
LIN {X 0,Y 149.84,Z 176.009,A -85,B 0,C 180,E1 -24999.073,E2 -24999.073} C_VEL
LIN {X 0,Y 141.334,Z 160.886,A -85,B 0,C 180,E1 -25003.94,E2 -25003.94} C_VEL
LIN {X 0,Y 136.473,Z 152.919,A -85,B 0,C 180,E1 -25007.004,E2 -25007.004} C_VEL
LIN {X 0,Y 133.965,Z 148.728,A -85,B 0,C 180,E1 -25008.706,E2 -25008.706} C_VEL
LIN {X 0,Y 131.911,Z 145.124,A -85,B 0,C 180,E1 -25010.22,E2 -25010.22} C_VEL
LIN {X 0,Y 130.126,Z 142.741,A -85,B 0,C 180,E1 -25011.459,E2 -25011.459} C_VEL
LIN {X 0,Y 129.52,Z 140.662,A -85,B 0,C 180,E1 -25012.204,E2 -25012.204} C_VEL
LIN {X 0,Y 130.087,Z 140.592,A -85,B 0,C 180,E1 -25020,E2 -25020} C_VEL
LIN {X 0,Y 129.527,Z 140.663,A -85,B 0,C 180,E1 -25029.368,E2 -25029.368} C_VEL
LIN {X 0,Y 129.391,Z 140.674,A -85,B 0,C 180,E1 -25032.549,E2 -25032.549} C_VEL
LIN {X 0,Y 129.156,Z 140.704,A -85,B 0,C 180,E1 -25039.056,E2 -25039.056} C_VEL
LIN {X 0,Y 129.105,Z 140.71,A -85,B 0,C 180,E1 -25042.399,E2 -25042.399} C_VEL
LIN {X 0,Y 129.032,Z 140.719,A -85,B 0,C 180,E1 -25049.374,E2 -25049.374} C_VEL
LIN {X 0,Y 128.978,Z 140.732,A -85,B 0,C 180,E1 -25055.184,E2 -25055.184} C_VEL
LIN {X 0,Y 128.932,Z 140.732,A -85,B 0,C 180,E1 -25060.853,E2 -25060.853} C_VEL
LIN {X 0,Y 128.925,Z 140.728,A -85,B 0,C 180,E1 -25065.126,E2 -25065.126} C_VEL
LIN {X 0,Y 128.991,Z 140.728,A -85,B 0,C 180,E1 -25069.71,E2 -25069.71} C_VEL
LIN {X 0,Y 128.995,Z 140.716,A -85,B 0,C 180,E1 -25074.81,E2 -25074.81} C_VEL
LIN {X 0,Y 129.032,Z 140.713,A -85,B 0,C 180,E1 -25080.649,E2 -25080.649} C_VEL
LIN {X 0,Y 129.135,Z 140.703,A -85,B 0,C 180,E1 -25087.609,E2 -25087.609} C_VEL
LIN {X 0,Y 129.179,Z 140.704,A -85,B 0,C 180,E1 -25090.95,E2 -25090.95} C_VEL
LIN {X 0,Y 129.417,Z 140.676,A -85,B 0,C 180,E1 -25097.822,E2 -25097.822} C_VEL
LIN {X 0,Y 129.524,Z 140.656,A -85,B 0,C 180,E1 -25100.634,E2 -25100.634} C_VEL
LIN {X 0,Y 130.091,Z 140.591,A -85,B 0,C 180,E1 -25110.002,E2 -25110.002} C_VEL
LIN {X 0,Y 129.533,Z 140.658,A -85,B 0,C 180,E1 -25119.37,E2 -25119.37} C_VEL
LIN {X 0,Y 129.452,Z 140.657,A -85,B 0,C 180,E1 -25120.932,E2 -25120.932} C_VEL
LIN {X 0,Y 130.388,Z 143.372,A -85,B 0,C 180,E1 -25121.837,E2 -25121.837} C_VEL
LIN {X 0,Y 132.297,Z 145.993,A -85,B 0,C 180,E1 -25123.148,E2 -25123.148} C_VEL
LIN {X 0,Y 134.306,Z 149.407,A -85,B 0,C 180,E1 -25124.588,E2 -25124.588} C_VEL
LIN {X 0,Y 139.773,Z 158.443,A -85,B 0,C 180,E1 -25128.14,E2 -25128.14} C_VEL
LIN {X 0,Y 147.172,Z 171.361,A -85,B 0,C 180,E1 -25132.461,E2 -25132.461} C_VEL
LIN {X 0,Y 156.24,Z 188.995,A -85,B 0,C 180,E1 -25137.242,E2 -25137.242} C_VEL
LIN {X 0,Y 165.378,Z 208.309,A -85,B 0,C 180,E1 -25141.552,E2 -25141.552} C_VEL
LIN {X 0,Y 171.96,Z 222.829,A -85,B 0,C 180,E1 -25144.379,E2 -25144.379} C_VEL
LIN {X 0,Y 158.599,Z 317.478,A -85,B 0,C 180,E1 -25150.879,E2 -25150.879} C_VEL
LIN {X 0,Y 155.387,Z 336.898,A -85,B 0,C 180,E1 -25152.833,E2 -25152.833} C_VEL
LIN {X 0,Y 151.698,Z 355.46,A -85,B 0,C 180,E1 -25155.282,E2 -25155.282} C_VEL
LIN {X 0,Y 147.671,Z 372.993,A -85,B 0,C 180,E1 -25158.218,E2 -25158.218} C_VEL
LIN {X 0,Y 143.463,Z 389.568,A -85,B 0,C 180,E1 -25161.706,E2 -25161.706} C_VEL
LIN {X 0,Y 139.34,Z 405.446,A -85,B 0,C 180,E1 -25165.866,E2 -25165.866} C_VEL
LIN {X 0,Y 135.589,Z 419.817,A -85,B 0,C 180,E1 -25170.5,E2 -25170.5} C_VEL
LIN {X 0,Y 132.77,Z 431.286,A -85,B 0,C 180,E1 -25174.946,E2 -25174.946} C_VEL
LIN {X 0,Y 130.331,Z 442.834,A -85,B 0,C 180,E1 -25180.304,E2 -25180.304} C_VEL
LIN {X 0,Y 128.451,Z 453.996,A -85,B 0,C 180,E1 -25186.554,E2 -25186.554} C_VEL
LIN {X 0,Y 127.688,Z 461.609,A -85,B 0,C 180,E1 -25191.571,E2 -25191.571} C_VEL
LIN {X 0,Y 127.344,Z 468.448,A -85,B 0,C 180,E1 -25196.836,E2 -25196.836} C_VEL
LIN {X 0,Y 127.641,Z 475.476,A -85,B 0,C 180,E1 -25203.156,E2 -25203.156} C_VEL
LIN {X 0,Y 128.693,Z 481.244,A -85,B 0,C 180,E1 -25209.429,E2 -25209.429} C_VEL
LIN {X 0,Y 131.603,Z 487.178,A -85,B 0,C 180,E1 -25217.08,E2 -25217.08} C_VEL
LIN {X 0,Y 136.613,Z 491.852,A -85,B 0,C 180,E1 -25224.302,E2 -25224.302} C_VEL
LIN {X 0,Y 145.273,Z 495.957,A -85,B 0,C 180,E1 -25232.151,E2 -25232.151} C_VEL
LIN {X 0,Y 152.6,Z 497.924,A -85,B 0,C 180,E1 -25236.778,E2 -25236.778} C_VEL
LIN {X 0,Y 161.984,Z 499.312,A -85,B 0,C 180,E1 -25241.272,E2 -25241.272} C_VEL
LIN {X 0,Y 161.245,Z 499.607,A -85,B 0,C 180,E1 -25242.184,E2 -25242.184} C_VEL
LIN {X 0,Y 148.534,Z 501.007,A -85,B 0,C 180,E1 -25248.513,E2 -25248.513} C_VEL
LIN {X 0,Y 138.524,Z 501.319,A -85,B 0,C 180,E1 -25256.074,E2 -25256.074} C_VEL
LIN {X 0,Y 131.862,Z 500.337,A -85,B 0,C 180,E1 -25264.759,E2 -25264.759} C_VEL
LIN {X 0,Y 129.371,Z 498.922,A -85,B 0,C 180,E1 -25270.975,E2 -25270.975} C_VEL
LIN {X 0,Y 128.555,Z 495.784,A -85,B 0,C 180,E1 -25279.749,E2 -25279.749} C_VEL
LIN {X 0,Y 129.041,Z 493.829,A -85,B 0,C 180,E1 -25283.744,E2 -25283.744} C_VEL
LIN {X 0,Y 129.684,Z 491.915,A -85,B 0,C 180,E1 -25286.891,E2 -25286.891} C_VEL
LIN {X 0,Y 129.953,Z 489.534,A -85,B 0,C 180,E1 -25289.998,E2 -25289.998} C_VEL
LIN {X 0,Y 129.635,Z 484.939,A -85,B 0,C 180,E1 -25294.662,E2 -25294.662} C_VEL
LIN {X 0,Y 129.4,Z 476.994,A -85,B 0,C 180,E1 -25301.086,E2 -25301.086} C_VEL
LIN {X 0,Y 129.919,Z 468.869,A -85,B 0,C 180,E1 -25306.497,E2 -25306.497} C_VEL
LIN {X 0,Y 131.251,Z 458.888,A -85,B 0,C 180,E1 -25312.011,E2 -25312.011} C_VEL
LIN {X 0,Y 133.534,Z 447.838,A -85,B 0,C 180,E1 -25317.092,E2 -25317.092} C_VEL
LIN {X 0,Y 136.834,Z 434.365,A -85,B 0,C 180,E1 -25322.197,E2 -25322.197} C_VEL
LIN {X 0,Y 140.607,Z 420.089,A -85,B 0,C 180,E1 -25326.567,E2 -25326.567} C_VEL
LIN {X 0,Y 141.929,Z 415.056,A -85,B 0,C 180,E1 -25327.908,E2 -25327.908} C_VEL
LIN {X 0,Y 142.533,Z 410.162,A -85,B 0,C 180,E1 -25329.158,E2 -25329.158} C_VEL
LIN {X 0,Y 141.402,Z 393.156,A -85,B 0,C 180,E1 -25333.259,E2 -25333.259} C_VEL
LIN {X 0,Y 142.072,Z 387.788,A -85,B 0,C 180,E1 -25334.326,E2 -25334.326} C_VEL
LIN {X 0,Y 146.25,Z 370.414,A -85,B 0,C 180,E1 -25337.128,E2 -25337.128} C_VEL
LIN {X 0,Y 150.042,Z 352.843,A -85,B 0,C 180,E1 -25339.305,E2 -25339.305} C_VEL
LIN {X 0,Y 152.967,Z 335.516,A -85,B 0,C 180,E1 -25340.961,E2 -25340.961} C_VEL
LIN {X 0,Y 167.747,Z 236.304,A -85,B 0,C 180,E1 -25348.003,E2 -25348.003} C_VEL
LIN {X 0,Y 158.652,Z 212.944,A -85,B 0,C 180,E1 -25352.416,E2 -25352.416} C_VEL
LIN {X 0,Y 150.611,Z 193.316,A -85,B 0,C 180,E1 -25356.782,E2 -25356.782} C_VEL
LIN {X 0,Y 144.791,Z 180.112,A -85,B 0,C 180,E1 -25360.192,E2 -25360.192} C_VEL
LIN {X 0,Y 136.836,Z 165.721,A -85,B 0,C 180,E1 -25365.02,E2 -25365.02} C_VEL
LIN {X 0,Y 129.785,Z 153.814,A -85,B 0,C 180,E1 -25369.864,E2 -25369.864} C_VEL
LIN {X 0,Y 127.748,Z 150.425,A -85,B 0,C 180,E1 -25371.385,E2 -25371.385} C_VEL
LIN {X 0,Y 125.673,Z 147.007,A -85,B 0,C 180,E1 -25373.024,E2 -25373.024} C_VEL
LIN {X 0,Y 124.714,Z 145.858,A -85,B 0,C 180,E1 -25373.732,E2 -25373.732} C_VEL
LIN {X 0,Y 123.039,Z 143.493,A -85,B 0,C 180,E1 -25375.085,E2 -25375.085} C_VEL
LIN {X 0,Y 122.535,Z 141.513,A -85,B 0,C 180,E1 -25375.889,E2 -25375.889} C_VEL
LIN {X 0,Y 123.041,Z 141.47,A -85,B 0,C 180,E1 -25380,E2 -25380} C_VEL
LIN {X 0,Y 122.421,Z 141.538,A -85,B 0,C 180,E1 -25387.203,E2 -25387.203} C_VEL
LIN {X 0,Y 122.361,Z 141.549,A -85,B 0,C 180,E1 -25392.479,E2 -25392.479} C_VEL
LIN {X 0,Y 122.114,Z 141.578,A -85,B 0,C 180,E1 -25396.724,E2 -25396.724} C_VEL
LIN {X 0,Y 122.02,Z 141.589,A -85,B 0,C 180,E1 -25402.851,E2 -25402.851} C_VEL
LIN {X 0,Y 121.954,Z 141.607,A -85,B 0,C 180,E1 -25407.454,E2 -25407.454} C_VEL
LIN {X 0,Y 121.907,Z 141.599,A -85,B 0,C 180,E1 -25411.256,E2 -25411.256} C_VEL
LIN {X 0,Y 121.895,Z 141.611,A -85,B 0,C 180,E1 -25416.182,E2 -25416.182} C_VEL
LIN {X 0,Y 121.87,Z 141.615,A -85,B 0,C 180,E1 -25421.441,E2 -25421.441} C_VEL
LIN {X 0,Y 121.909,Z 141.606,A -85,B 0,C 180,E1 -25428.543,E2 -25428.543} C_VEL
LIN {X 0,Y 121.948,Z 141.593,A -85,B 0,C 180,E1 -25434.811,E2 -25434.811} C_VEL
LIN {X 0,Y 121.941,Z 141.601,A -85,B 0,C 180,E1 -25439.828,E2 -25439.828} C_VEL
LIN {X 0,Y 122.068,Z 141.586,A -85,B 0,C 180,E1 -25447.102,E2 -25447.102} C_VEL
LIN {X 0,Y 122.124,Z 141.584,A -85,B 0,C 180,E1 -25453.28,E2 -25453.28} C_VEL
LIN {X 0,Y 122.364,Z 141.554,A -85,B 0,C 180,E1 -25457.528,E2 -25457.528} C_VEL
LIN {X 0,Y 122.452,Z 141.539,A -85,B 0,C 180,E1 -25460.088,E2 -25460.088} C_VEL
LIN {X 0,Y 122.61,Z 141.517,A -85,B 0,C 180,E1 -25466.716,E2 -25466.716} C_VEL
LIN {X 0,Y 123.045,Z 141.469,A -85,B 0,C 180,E1 -25470.002,E2 -25470.002} C_VEL
LIN {X 0,Y 122.45,Z 141.576,A -85,B 0,C 180,E1 -25477.318,E2 -25477.318} C_VEL
LIN {X 0,Y 123.33,Z 144.199,A -85,B 0,C 180,E1 -25478.296,E2 -25478.296} C_VEL
LIN {X 0,Y 125.555,Z 146.894,A -85,B 0,C 180,E1 -25479.961,E2 -25479.961} C_VEL
LIN {X 0,Y 127.497,Z 150.261,A -85,B 0,C 180,E1 -25481.535,E2 -25481.535} C_VEL
LIN {X 0,Y 134.192,Z 161.387,A -85,B 0,C 180,E1 -25486.313,E2 -25486.313} C_VEL
LIN {X 0,Y 141.419,Z 174.091,A -85,B 0,C 180,E1 -25490.841,E2 -25490.841} C_VEL
LIN {X 0,Y 149.182,Z 189.268,A -85,B 0,C 180,E1 -25495.249,E2 -25495.249} C_VEL
LIN {X 0,Y 157.25,Z 206.129,A -85,B 0,C 180,E1 -25499.357,E2 -25499.357} C_VEL
LIN {X 0,Y 165.619,Z 224.822,A -85,B 0,C 180,E1 -25503.232,E2 -25503.232} C_VEL
LIN {X 0,Y 151.946,Z 318.547,A -85,B 0,C 180,E1 -25509.935,E2 -25509.935} C_VEL
LIN {X 0,Y 148.699,Z 337.291,A -85,B 0,C 180,E1 -25511.892,E2 -25511.892} C_VEL
LIN {X 0,Y 145.013,Z 355.354,A -85,B 0,C 180,E1 -25514.369,E2 -25514.369} C_VEL
LIN {X 0,Y 141.075,Z 372.055,A -85,B 0,C 180,E1 -25517.253,E2 -25517.253} C_VEL
LIN {X 0,Y 136.716,Z 388.842,A -85,B 0,C 180,E1 -25520.879,E2 -25520.879} C_VEL
LIN {X 0,Y 132.439,Z 404.805,A -85,B 0,C 180,E1 -25525.218,E2 -25525.218} C_VEL
LIN {X 0,Y 128.589,Z 419.3,A -85,B 0,C 180,E1 -25530.084,E2 -25530.084} C_VEL
LIN {X 0,Y 125.481,Z 431.736,A -85,B 0,C 180,E1 -25535.161,E2 -25535.161} C_VEL
LIN {X 0,Y 123.094,Z 443.241,A -85,B 0,C 180,E1 -25540.834,E2 -25540.834} C_VEL
LIN {X 0,Y 121.207,Z 454.33,A -85,B 0,C 180,E1 -25547.441,E2 -25547.441} C_VEL
LIN {X 0,Y 120.502,Z 462.633,A -85,B 0,C 180,E1 -25553.301,E2 -25553.301} C_VEL
LIN {X 0,Y 120.45,Z 470.634,A -85,B 0,C 180,E1 -25560,E2 -25560} C_VEL
LIN {X 0,Y 121.163,Z 477.269,A -85,B 0,C 180,E1 -25566.661,E2 -25566.661} C_VEL
LIN {X 0,Y 123.335,Z 484.094,A -85,B 0,C 180,E1 -25574.858,E2 -25574.858} C_VEL
LIN {X 0,Y 127.819,Z 489.53,A -85,B 0,C 180,E1 -25582.636,E2 -25582.636} C_VEL
LIN {X 0,Y 132.942,Z 493.089,A -85,B 0,C 180,E1 -25588.41,E2 -25588.41} C_VEL
LIN {X 0,Y 142.983,Z 497.082,A -85,B 0,C 180,E1 -25596.145,E2 -25596.145} C_VEL
LIN {X 0,Y 152.449,Z 499.209,A -85,B 0,C 180,E1 -25601.118,E2 -25601.118} C_VEL
LIN {X 0,Y 151.897,Z 499.519,A -85,B 0,C 180,E1 -25602.241,E2 -25602.241} C_VEL
LIN {X 0,Y 139.16,Z 500.16,A -85,B 0,C 180,E1 -25609.247,E2 -25609.247} C_VEL
LIN {X 0,Y 129.92,Z 499.755,A -85,B 0,C 180,E1 -25617.249,E2 -25617.249} C_VEL
LIN {X 0,Y 123.95,Z 497.999,A -85,B 0,C 180,E1 -25626.613,E2 -25626.613} C_VEL
LIN {X 0,Y 121.801,Z 494.804,A -85,B 0,C 180,E1 -25636.653,E2 -25636.653} C_VEL
LIN {X 0,Y 122.293,Z 491.643,A -85,B 0,C 180,E1 -25643.398,E2 -25643.398} C_VEL
LIN {X 0,Y 122.94,Z 489.68,A -85,B 0,C 180,E1 -25646.721,E2 -25646.721} C_VEL
LIN {X 0,Y 123.163,Z 487.196,A -85,B 0,C 180,E1 -25649.998,E2 -25649.998} C_VEL
LIN {X 0,Y 122.783,Z 482.339,A -85,B 0,C 180,E1 -25654.923,E2 -25654.923} C_VEL
LIN {X 0,Y 122.57,Z 475.094,A -85,B 0,C 180,E1 -25660.893,E2 -25660.893} C_VEL
LIN {X 0,Y 123.216,Z 465.46,A -85,B 0,C 180,E1 -25667.422,E2 -25667.422} C_VEL
LIN {X 0,Y 124.766,Z 455.056,A -85,B 0,C 180,E1 -25673.22,E2 -25673.22} C_VEL
LIN {X 0,Y 127.261,Z 443.684,A -85,B 0,C 180,E1 -25678.505,E2 -25678.505} C_VEL
LIN {X 0,Y 130.555,Z 430.601,A -85,B 0,C 180,E1 -25683.486,E2 -25683.486} C_VEL
LIN {X 0,Y 134.411,Z 416.524,A -85,B 0,C 180,E1 -25687.828,E2 -25687.828} C_VEL
LIN {X 0,Y 138.64,Z 400.9,A -85,B 0,C 180,E1 -25691.706,E2 -25691.706} C_VEL
LIN {X 0,Y 142.072,Z 387.788,A -85,B 0,C 180,E1 -25694.326,E2 -25694.326} C_VEL
LIN {X 0,Y 142.691,Z 382.521,A -85,B 0,C 180,E1 -25695.336,E2 -25695.336} C_VEL
LIN {X 0,Y 141.371,Z 364.595,A -85,B 0,C 180,E1 -25698.724,E2 -25698.724} C_VEL
LIN {X 0,Y 142.035,Z 358.987,A -85,B 0,C 180,E1 -25699.532,E2 -25699.532} C_VEL
LIN {X 0,Y 145.466,Z 341.504,A -85,B 0,C 180,E1 -25701.448,E2 -25701.448} C_VEL
LIN {X 0,Y 158.563,Z 256.074,A -85,B 0,C 180,E1 -25707.967,E2 -25707.967} C_VEL
LIN {X 0,Y 161.405,Z 237.97,A -85,B 0,C 180,E1 -25709.195,E2 -25709.195} C_VEL
LIN {X 0,Y 152.677,Z 215.23,A -85,B 0,C 180,E1 -25713.701,E2 -25713.701} C_VEL
LIN {X 0,Y 144.866,Z 195.988,A -85,B 0,C 180,E1 -25718.196,E2 -25718.196} C_VEL
LIN {X 0,Y 139.84,Z 184.363,A -85,B 0,C 180,E1 -25721.347,E2 -25721.347} C_VEL
LIN {X 0,Y 132.17,Z 170.267,A -85,B 0,C 180,E1 -25726.251,E2 -25726.251} C_VEL
LIN {X 0,Y 125.251,Z 158.329,A -85,B 0,C 180,E1 -25731.327,E2 -25731.327} C_VEL
LIN {X 0,Y 123.124,Z 154.893,A -85,B 0,C 180,E1 -25733.033,E2 -25733.033} C_VEL
LIN {X 0,Y 121.098,Z 151.642,A -85,B 0,C 180,E1 -25734.714,E2 -25734.714} C_VEL
LIN {X 0,Y 118.934,Z 148.309,A -85,B 0,C 180,E1 -25736.613,E2 -25736.613} C_VEL
LIN {X 0,Y 118.313,Z 147.11,A -85,B 0,C 180,E1 -25737.234,E2 -25737.234} C_VEL
LIN {X 0,Y 116.537,Z 144.773,A -85,B 0,C 180,E1 -25738.813,E2 -25738.813} C_VEL
LIN {X 0,Y 115.939,Z 142.355,A -85,B 0,C 180,E1 -25739.783,E2 -25739.783} C_VEL
LIN {X 0,Y 115.387,Z 142.417,A -85,B 0,C 180,E1 -25747.095,E2 -25747.095} C_VEL
LIN {X 0,Y 115.283,Z 142.431,A -85,B 0,C 180,E1 -25752.743,E2 -25752.743} C_VEL
LIN {X 0,Y 115.015,Z 142.46,A -85,B 0,C 180,E1 -25757.79,E2 -25757.79} C_VEL
LIN {X 0,Y 114.943,Z 142.467,A -85,B 0,C 180,E1 -25763.493,E2 -25763.493} C_VEL
LIN {X 0,Y 114.864,Z 142.476,A -85,B 0,C 180,E1 -25771.068,E2 -25771.068} C_VEL
LIN {X 0,Y 114.784,Z 142.487,A -85,B 0,C 180,E1 -25777.755,E2 -25777.755} C_VEL
LIN {X 0,Y 114.787,Z 142.5,A -85,B 0,C 180,E1 -25782.72,E2 -25782.72} C_VEL
LIN {X 0,Y 114.82,Z 142.483,A -85,B 0,C 180,E1 -25787.681,E2 -25787.681} C_VEL
LIN {X 0,Y 114.825,Z 142.483,A -85,B 0,C 180,E1 -25792.72,E2 -25792.72} C_VEL
LIN {X 0,Y 114.868,Z 142.487,A -85,B 0,C 180,E1 -25798.934,E2 -25798.934} C_VEL
LIN {X 0,Y 114.965,Z 142.474,A -85,B 0,C 180,E1 -25806.488,E2 -25806.488} C_VEL
LIN {X 0,Y 115.028,Z 142.47,A -85,B 0,C 180,E1 -25812.215,E2 -25812.215} C_VEL
LIN {X 0,Y 115.285,Z 142.434,A -85,B 0,C 180,E1 -25817.263,E2 -25817.263} C_VEL
LIN {X 0,Y 115.395,Z 142.42,A -85,B 0,C 180,E1 -25823.006,E2 -25823.006} C_VEL
LIN {X 0,Y 115.997,Z 142.347,A -85,B 0,C 180,E1 -25830.002,E2 -25830.002} C_VEL
LIN {X 0,Y 115.569,Z 142.377,A -85,B 0,C 180,E1 -25833.162,E2 -25833.162} C_VEL
LIN {X 0,Y 116.347,Z 144.992,A -85,B 0,C 180,E1 -25834.224,E2 -25834.224} C_VEL
LIN {X 0,Y 118.114,Z 147.122,A -85,B 0,C 180,E1 -25835.765,E2 -25835.765} C_VEL
LIN {X 0,Y 118.791,Z 148.146,A -85,B 0,C 180,E1 -25836.371,E2 -25836.371} C_VEL
LIN {X 0,Y 120.841,Z 151.369,A -85,B 0,C 180,E1 -25838.194,E2 -25838.194} C_VEL
LIN {X 0,Y 121.867,Z 152.886,A -85,B 0,C 180,E1 -25839.044,E2 -25839.044} C_VEL
LIN {X 0,Y 129.129,Z 165.132,A -85,B 0,C 180,E1 -25844.676,E2 -25844.676} C_VEL
LIN {X 0,Y 135.183,Z 175.974,A -85,B 0,C 180,E1 -25848.787,E2 -25848.787} C_VEL
LIN {X 0,Y 141.06,Z 187.235,A -85,B 0,C 180,E1 -25852.426,E2 -25852.426} C_VEL
LIN {X 0,Y 148.9,Z 203.531,A -85,B 0,C 180,E1 -25856.829,E2 -25856.829} C_VEL
LIN {X 0,Y 156.876,Z 221.216,A -85,B 0,C 180,E1 -25860.872,E2 -25860.872} C_VEL
LIN {X 0,Y 159.356,Z 226.807,A -85,B 0,C 180,E1 -25862.039,E2 -25862.039} C_VEL
LIN {X 0,Y 145.457,Z 318.423,A -85,B 0,C 180,E1 -25868.822,E2 -25868.822} C_VEL
LIN {X 0,Y 141.937,Z 338.135,A -85,B 0,C 180,E1 -25870.965,E2 -25870.965} C_VEL
LIN {X 0,Y 138.121,Z 356.051,A -85,B 0,C 180,E1 -25873.524,E2 -25873.524} C_VEL
LIN {X 0,Y 134.078,Z 372.618,A -85,B 0,C 180,E1 -25876.53,E2 -25876.53} C_VEL
LIN {X 0,Y 129.552,Z 389.582,A -85,B 0,C 180,E1 -25880.4,E2 -25880.4} C_VEL
LIN {X 0,Y 125.254,Z 405.257,A -85,B 0,C 180,E1 -25884.891,E2 -25884.891} C_VEL
LIN {X 0,Y 121.293,Z 419.888,A -85,B 0,C 180,E1 -25890.113,E2 -25890.113} C_VEL
LIN {X 0,Y 118.208,Z 432.092,A -85,B 0,C 180,E1 -25895.406,E2 -25895.406} C_VEL
LIN {X 0,Y 115.81,Z 443.521,A -85,B 0,C 180,E1 -25901.421,E2 -25901.421} C_VEL
LIN {X 0,Y 114.116,Z 454.618,A -85,B 0,C 180,E1 -25908.454,E2 -25908.454} C_VEL
LIN {X 0,Y 113.468,Z 462.889,A -85,B 0,C 180,E1 -25914.669,E2 -25914.669} C_VEL
LIN {X 0,Y 113.58,Z 470.823,A -85,B 0,C 180,E1 -25921.773,E2 -25921.773} C_VEL
LIN {X 0,Y 114.55,Z 477.466,A -85,B 0,C 180,E1 -25928.823,E2 -25928.823} C_VEL
LIN {X 0,Y 117.354,Z 484.299,A -85,B 0,C 180,E1 -25937.423,E2 -25937.423} C_VEL
LIN {X 0,Y 121.326,Z 488.813,A -85,B 0,C 180,E1 -25943.921,E2 -25943.921} C_VEL
LIN {X 0,Y 129.969,Z 494.246,A -85,B 0,C 180,E1 -25952.734,E2 -25952.734} C_VEL
LIN {X 0,Y 141.482,Z 498.171,A -85,B 0,C 180,E1 -25960.222,E2 -25960.222} C_VEL
LIN {X 0,Y 142.931,Z 498.549,A -85,B 0,C 180,E1 -25960.956,E2 -25960.956} C_VEL
LIN {X 0,Y 143.407,Z 498.859,A -85,B 0,C 180,E1 -25961.933,E2 -25961.933} C_VEL
LIN {X 0,Y 130.455,Z 498.818,A -85,B 0,C 180,E1 -25969.721,E2 -25969.721} C_VEL
LIN {X 0,Y 121.469,Z 497.692,A -85,B 0,C 180,E1 -25978.617,E2 -25978.617} C_VEL
LIN {X 0,Y 116.306,Z 495.182,A -85,B 0,C 180,E1 -25988.74,E2 -25988.74} C_VEL
LIN {X 0,Y 115.096,Z 491.962,A -85,B 0,C 180,E1 -25997.684,E2 -25997.684} C_VEL
LIN {X 0,Y 115.853,Z 488.363,A -85,B 0,C 180,E1 -26004.777,E2 -26004.777} C_VEL
LIN {X 0,Y 116.43,Z 486.117,A -85,B 0,C 180,E1 -26008.268,E2 -26008.268} C_VEL
LIN {X 0,Y 116.292,Z 483.104,A -85,B 0,C 180,E1 -26011.729,E2 -26011.729} C_VEL
LIN {X 0,Y 115.767,Z 476.561,A -85,B 0,C 180,E1 -26017.848,E2 -26017.848} C_VEL
LIN {X 0,Y 115.907,Z 468.601,A -85,B 0,C 180,E1 -26024.034,E2 -26024.034} C_VEL
LIN {X 0,Y 116.922,Z 458.947,A -85,B 0,C 180,E1 -26030.217,E2 -26030.217} C_VEL
LIN {X 0,Y 119.07,Z 447.611,A -85,B 0,C 180,E1 -26036.272,E2 -26036.272} C_VEL
LIN {X 0,Y 122.384,Z 434.208,A -85,B 0,C 180,E1 -26042.083,E2 -26042.083} C_VEL
LIN {X 0,Y 126.388,Z 419.451,A -85,B 0,C 180,E1 -26047.206,E2 -26047.206} C_VEL
LIN {X 0,Y 130.791,Z 403.78,A -85,B 0,C 180,E1 -26051.522,E2 -26051.522} C_VEL
LIN {X 0,Y 135.311,Z 387.04,A -85,B 0,C 180,E1 -26055.14,E2 -26055.14} C_VEL
LIN {X 0,Y 139.487,Z 370.139,A -85,B 0,C 180,E1 -26057.999,E2 -26057.999} C_VEL
LIN {X 0,Y 142.035,Z 358.987,A -85,B 0,C 180,E1 -26059.532,E2 -26059.532} C_VEL
LIN {X 0,Y 142.611,Z 353.424,A -85,B 0,C 180,E1 -26060.297,E2 -26060.297} C_VEL
LIN {X 0,Y 141.617,Z 344.187,A -85,B 0,C 180,E1 -26061.716,E2 -26061.716} C_VEL
LIN {X 0,Y 140.485,Z 334.842,A -85,B 0,C 180,E1 -26063.049,E2 -26063.049} C_VEL
LIN {X 0,Y 140.826,Z 329.1,A -85,B 0,C 180,E1 -26063.641,E2 -26063.641} C_VEL
LIN {X 0,Y 155.099,Z 239.822,A -85,B 0,C 180,E1 -26070.413,E2 -26070.413} C_VEL
LIN {X 0,Y 147.542,Z 219.71,A -85,B 0,C 180,E1 -26074.559,E2 -26074.559} C_VEL
LIN {X 0,Y 139.877,Z 200.322,A -85,B 0,C 180,E1 -26079.246,E2 -26079.246} C_VEL
LIN {X 0,Y 134.855,Z 188.479,A -85,B 0,C 180,E1 -26082.58,E2 -26082.58} C_VEL
LIN {X 0,Y 127.537,Z 174.78,A -85,B 0,C 180,E1 -26087.578,E2 -26087.578} C_VEL
LIN {X 0,Y 119.992,Z 161.317,A -85,B 0,C 180,E1 -26093.567,E2 -26093.567} C_VEL
LIN {X 0,Y 116.975,Z 156.736,A -85,B 0,C 180,E1 -26096.188,E2 -26096.188} C_VEL
LIN {X 0,Y 114.225,Z 152.354,A -85,B 0,C 180,E1 -26098.788,E2 -26098.788} C_VEL
LIN {X 0,Y 112.451,Z 149.252,A -85,B 0,C 180,E1 -26100.668,E2 -26100.668} C_VEL
LIN {X 0,Y 111.939,Z 148.336,A -85,B 0,C 180,E1 -26101.234,E2 -26101.234} C_VEL
LIN {X 0,Y 109.508,Z 146.185,A -85,B 0,C 180,E1 -26103.565,E2 -26103.565} C_VEL
LIN {X 0,Y 108.468,Z 143.77,A -85,B 0,C 180,E1 -26104.995,E2 -26104.995} C_VEL
LIN {X 0,Y 108.379,Z 143.29,A -85,B 0,C 180,E1 -26105.349,E2 -26105.349} C_VEL
LIN {X 0,Y 108.29,Z 143.299,A -85,B 0,C 180,E1 -26111.228,E2 -26111.228} C_VEL
LIN {X 0,Y 107.905,Z 143.349,A -85,B 0,C 180,E1 -26119.006,E2 -26119.006} C_VEL
LIN {X 0,Y 107.855,Z 143.349,A -85,B 0,C 180,E1 -26124.187,E2 -26124.187} C_VEL
LIN {X 0,Y 107.788,Z 143.358,A -85,B 0,C 180,E1 -26132.051,E2 -26132.051} C_VEL
LIN {X 0,Y 107.691,Z 143.368,A -85,B 0,C 180,E1 -26138.456,E2 -26138.456} C_VEL
LIN {X 0,Y 107.691,Z 143.367,A -85,B 0,C 180,E1 -26145.879,E2 -26145.879} C_VEL
LIN {X 0,Y 107.723,Z 143.375,A -85,B 0,C 180,E1 -26151.527,E2 -26151.527} C_VEL
LIN {X 0,Y 107.806,Z 143.367,A -85,B 0,C 180,E1 -26158.568,E2 -26158.568} C_VEL
LIN {X 0,Y 107.931,Z 143.346,A -85,B 0,C 180,E1 -26167.005,E2 -26167.005} C_VEL
LIN {X 0,Y 108.043,Z 143.328,A -85,B 0,C 180,E1 -26174.921,E2 -26174.921} C_VEL
LIN {X 0,Y 108.304,Z 143.307,A -85,B 0,C 180,E1 -26178.777,E2 -26178.777} C_VEL
LIN {X 0,Y 108.462,Z 143.279,A -85,B 0,C 180,E1 -26186.287,E2 -26186.287} C_VEL
LIN {X 0,Y 108.698,Z 143.461,A -85,B 0,C 180,E1 -26188.266,E2 -26188.266} C_VEL
LIN {X 0,Y 109.815,Z 145.965,A -85,B 0,C 180,E1 -26189.773,E2 -26189.773} C_VEL
LIN {X 0,Y 111.948,Z 148.705,A -85,B 0,C 180,E1 -26191.981,E2 -26191.981} C_VEL
LIN {X 0,Y 113.556,Z 151.792,A -85,B 0,C 180,E1 -26193.773,E2 -26193.773} C_VEL
LIN {X 0,Y 115.244,Z 154.109,A -85,B 0,C 180,E1 -26195.36,E2 -26195.36} C_VEL
LIN {X 0,Y 118.059,Z 158.523,A -85,B 0,C 180,E1 -26197.92,E2 -26197.92} C_VEL
LIN {X 0,Y 122.695,Z 166.438,A -85,B 0,C 180,E1 -26201.829,E2 -26201.829} C_VEL
LIN {X 0,Y 128.739,Z 177.208,A -85,B 0,C 180,E1 -26206.355,E2 -26206.355} C_VEL
LIN {X 0,Y 133.654,Z 186.647,A -85,B 0,C 180,E1 -26209.712,E2 -26209.712} C_VEL
LIN {X 0,Y 141.72,Z 203.17,A -85,B 0,C 180,E1 -26214.659,E2 -26214.659} C_VEL
LIN {X 0,Y 150.336,Z 222.455,A -85,B 0,C 180,E1 -26219.382,E2 -26219.382} C_VEL
LIN {X 0,Y 153.098,Z 228.945,A -85,B 0,C 180,E1 -26220.787,E2 -26220.787} C_VEL
LIN {X 0,Y 138.916,Z 318.693,A -85,B 0,C 180,E1 -26227.67,E2 -26227.67} C_VEL
LIN {X 0,Y 135.477,Z 337.553,A -85,B 0,C 180,E1 -26229.788,E2 -26229.788} C_VEL
LIN {X 0,Y 131.296,Z 356.541,A -85,B 0,C 180,E1 -26232.607,E2 -26232.607} C_VEL
LIN {X 0,Y 127.305,Z 372.395,A -85,B 0,C 180,E1 -26235.59,E2 -26235.59} C_VEL
LIN {X 0,Y 122.467,Z 389.918,A -85,B 0,C 180,E1 -26239.789,E2 -26239.789} C_VEL
LIN {X 0,Y 118.075,Z 405.568,A -85,B 0,C 180,E1 -26244.526,E2 -26244.526} C_VEL
LIN {X 0,Y 114.178,Z 419.75,A -85,B 0,C 180,E1 -26249.877,E2 -26249.877} C_VEL
LIN {X 0,Y 110.534,Z 434.05,A -85,B 0,C 180,E1 -26256.585,E2 -26256.585} C_VEL
LIN {X 0,Y 108.221,Z 445.213,A -85,B 0,C 180,E1 -26263.008,E2 -26263.008} C_VEL
LIN {X 0,Y 106.96,Z 454.857,A -85,B 0,C 180,E1 -26269.642,E2 -26269.642} C_VEL
LIN {X 0,Y 106.467,Z 463.051,A -85,B 0,C 180,E1 -26276.215,E2 -26276.215} C_VEL
LIN {X 0,Y 106.806,Z 470.925,A -85,B 0,C 180,E1 -26283.772,E2 -26283.772} C_VEL
LIN {X 0,Y 108.098,Z 477.584,A -85,B 0,C 180,E1 -26291.247,E2 -26291.247} C_VEL
LIN {X 0,Y 111.6,Z 484.401,A -85,B 0,C 180,E1 -26300.265,E2 -26300.265} C_VEL
LIN {X 0,Y 117.607,Z 490.015,A -85,B 0,C 180,E1 -26308.559,E2 -26308.559} C_VEL
LIN {X 0,Y 127.73,Z 495.329,A -85,B 0,C 180,E1 -26317.246,E2 -26317.246} C_VEL
LIN {X 0,Y 134.406,Z 497.59,A -85,B 0,C 180,E1 -26321.232,E2 -26321.232} C_VEL
LIN {X 0,Y 133.352,Z 497.745,A -85,B 0,C 180,E1 -26322.45,E2 -26322.45} C_VEL
LIN {X 0,Y 121.573,Z 496.986,A -85,B 0,C 180,E1 -26330.511,E2 -26330.511} C_VEL
LIN {X 0,Y 113.069,Z 495.072,A -85,B 0,C 180,E1 -26340.48,E2 -26340.48} C_VEL
LIN {X 0,Y 108.997,Z 491.896,A -85,B 0,C 180,E1 -26351.19,E2 -26351.19} C_VEL
LIN {X 0,Y 108.519,Z 488.868,A -85,B 0,C 180,E1 -26358.794,E2 -26358.794} C_VEL
LIN {X 0,Y 109.599,Z 484.845,A -85,B 0,C 180,E1 -26366.321,E2 -26366.321} C_VEL
LIN {X 0,Y 109.784,Z 483.528,A -85,B 0,C 180,E1 -26368.163,E2 -26368.163} C_VEL
LIN {X 0,Y 109.528,Z 480.374,A -85,B 0,C 180,E1 -26371.836,E2 -26371.836} C_VEL
LIN {X 0,Y 108.972,Z 473.505,A -85,B 0,C 180,E1 -26378.341,E2 -26378.341} C_VEL
LIN {X 0,Y 109.207,Z 464.795,A -85,B 0,C 180,E1 -26385.135,E2 -26385.135} C_VEL
LIN {X 0,Y 110.339,Z 455.057,A -85,B 0,C 180,E1 -26391.482,E2 -26391.482} C_VEL
LIN {X 0,Y 112.796,Z 443.285,A -85,B 0,C 180,E1 -26397.835,E2 -26397.835} C_VEL
LIN {X 0,Y 116.134,Z 430.291,A -85,B 0,C 180,E1 -26403.516,E2 -26403.516} C_VEL
LIN {X 0,Y 120.482,Z 415.072,A -85,B 0,C 180,E1 -26408.831,E2 -26408.831} C_VEL
LIN {X 0,Y 125.169,Z 398.49,A -85,B 0,C 180,E1 -26413.343,E2 -26413.343} C_VEL
LIN {X 0,Y 129.329,Z 383.279,A -85,B 0,C 180,E1 -26416.618,E2 -26416.618} C_VEL
LIN {X 0,Y 133.806,Z 365.457,A -85,B 0,C 180,E1 -26419.602,E2 -26419.602} C_VEL
LIN {X 0,Y 137.848,Z 347.01,A -85,B 0,C 180,E1 -26421.916,E2 -26421.916} C_VEL
LIN {X 0,Y 140.826,Z 329.1,A -85,B 0,C 180,E1 -26423.641,E2 -26423.641} C_VEL
LIN {X 0,Y 141.156,Z 323.385,A -85,B 0,C 180,E1 -26424.215,E2 -26424.215} C_VEL
LIN {X 0,Y 138.774,Z 304.717,A -85,B 0,C 180,E1 -26426.797,E2 -26426.797} C_VEL
LIN {X 0,Y 139.047,Z 298.992,A -85,B 0,C 180,E1 -26427.403,E2 -26427.403} C_VEL
LIN {X 0,Y 148.846,Z 241.51,A -85,B 0,C 180,E1 -26431.72,E2 -26431.72} C_VEL
LIN {X 0,Y 140.71,Z 219.626,A -85,B 0,C 180,E1 -26436.519,E2 -26436.519} C_VEL
LIN {X 0,Y 133.53,Z 201.228,A -85,B 0,C 180,E1 -26441.284,E2 -26441.284} C_VEL
LIN {X 0,Y 129.718,Z 192.292,A -85,B 0,C 180,E1 -26444.001,E2 -26444.001} C_VEL
LIN {X 0,Y 122.544,Z 178.538,A -85,B 0,C 180,E1 -26449.252,E2 -26449.252} C_VEL
LIN {X 0,Y 115.775,Z 166.338,A -85,B 0,C 180,E1 -26455.03,E2 -26455.03} C_VEL
LIN {X 0,Y 113.155,Z 162.194,A -85,B 0,C 180,E1 -26457.453,E2 -26457.453} C_VEL
LIN {X 0,Y 110.285,Z 157.471,A -85,B 0,C 180,E1 -26460.426,E2 -26460.426} C_VEL
LIN {X 0,Y 108.375,Z 154.251,A -85,B 0,C 180,E1 -26462.556,E2 -26462.556} C_VEL
LIN {X 0,Y 105.938,Z 151.535,A -85,B 0,C 180,E1 -26465.202,E2 -26465.202} C_VEL
LIN {X 0,Y 104.841,Z 149.454,A -85,B 0,C 180,E1 -26466.685,E2 -26466.685} C_VEL
LIN {X 0,Y 102.46,Z 147.404,A -85,B 0,C 180,E1 -26469.501,E2 -26469.501} C_VEL
LIN {X 0,Y 101.314,Z 144.67,A -85,B 0,C 180,E1 -26471.504,E2 -26471.504} C_VEL
LIN {X 0,Y 101.21,Z 144.181,A -85,B 0,C 180,E1 -26471.897,E2 -26471.897} C_VEL
LIN {X 0,Y 100.815,Z 144.24,A -85,B 0,C 180,E1 -26480.4,E2 -26480.4} C_VEL
LIN {X 0,Y 100.771,Z 144.232,A -85,B 0,C 180,E1 -26484.96,E2 -26484.96} C_VEL
LIN {X 0,Y 100.693,Z 144.247,A -85,B 0,C 180,E1 -26493.123,E2 -26493.123} C_VEL
LIN {X 0,Y 100.641,Z 144.248,A -85,B 0,C 180,E1 -26499.816,E2 -26499.816} C_VEL
LIN {X 0,Y 100.659,Z 144.243,A -85,B 0,C 180,E1 -26505.721,E2 -26505.721} C_VEL
LIN {X 0,Y 100.661,Z 144.256,A -85,B 0,C 180,E1 -26511.074,E2 -26511.074} C_VEL
LIN {X 0,Y 100.7,Z 144.251,A -85,B 0,C 180,E1 -26516.877,E2 -26516.877} C_VEL
LIN {X 0,Y 100.785,Z 144.244,A -85,B 0,C 180,E1 -26525.27,E2 -26525.27} C_VEL
LIN {X 0,Y 100.834,Z 144.225,A -85,B 0,C 180,E1 -26529.608,E2 -26529.608} C_VEL
LIN {X 0,Y 101.198,Z 144.192,A -85,B 0,C 180,E1 -26537.977,E2 -26537.977} C_VEL
LIN {X 0,Y 101.26,Z 144.349,A -85,B 0,C 180,E1 -26541.521,E2 -26541.521} C_VEL
LIN {X 0,Y 102.36,Z 147.095,A -85,B 0,C 180,E1 -26543.473,E2 -26543.473} C_VEL
LIN {X 0,Y 104.532,Z 149.196,A -85,B 0,C 180,E1 -26546.147,E2 -26546.147} C_VEL
LIN {X 0,Y 105.458,Z 149.827,A -85,B 0,C 180,E1 -26547.128,E2 -26547.128} C_VEL
LIN {X 0,Y 108.495,Z 154.757,A -85,B 0,C 180,E1 -26550.814,E2 -26550.814} C_VEL
LIN {X 0,Y 110.676,Z 158.333,A -85,B 0,C 180,E1 -26553.188,E2 -26553.188} C_VEL
LIN {X 0,Y 114.267,Z 164.076,A -85,B 0,C 180,E1 -26556.735,E2 -26556.735} C_VEL
LIN {X 0,Y 120.522,Z 175.014,A -85,B 0,C 180,E1 -26562.202,E2 -26562.202} C_VEL
LIN {X 0,Y 127.511,Z 188.222,A -85,B 0,C 180,E1 -26567.522,E2 -26567.522} C_VEL
LIN {X 0,Y 134.647,Z 203.136,A -85,B 0,C 180,E1 -26572.346,E2 -26572.346} C_VEL
LIN {X 0,Y 142.117,Z 219.739,A -85,B 0,C 180,E1 -26576.826,E2 -26576.826} C_VEL
LIN {X 0,Y 146.797,Z 230.611,A -85,B 0,C 180,E1 -26579.387,E2 -26579.387} C_VEL
LIN {X 0,Y 132.119,Z 320.594,A -85,B 0,C 180,E1 -26586.602,E2 -26586.602} C_VEL
LIN {X 0,Y 128.568,Z 339.182,A -85,B 0,C 180,E1 -26588.834,E2 -26588.834} C_VEL
LIN {X 0,Y 124.529,Z 356.869,A -85,B 0,C 180,E1 -26591.601,E2 -26591.601} C_VEL
LIN {X 0,Y 120.238,Z 373.08,A -85,B 0,C 180,E1 -26594.8,E2 -26594.8} C_VEL
LIN {X 0,Y 115.429,Z 390.154,A -85,B 0,C 180,E1 -26599.116,E2 -26599.116} C_VEL
LIN {X 0,Y 110.879,Z 405.712,A -85,B 0,C 180,E1 -26604.104,E2 -26604.104} C_VEL
LIN {X 0,Y 107.165,Z 419.139,A -85,B 0,C 180,E1 -26609.452,E2 -26609.452} C_VEL
LIN {X 0,Y 103.689,Z 432.43,A -85,B 0,C 180,E1 -26616.003,E2 -26616.003} C_VEL
LIN {X 0,Y 101.573,Z 442.282,A -85,B 0,C 180,E1 -26621.858,E2 -26621.858} C_VEL
LIN {X 0,Y 100.034,Z 453.295,A -85,B 0,C 180,E1 -26629.619,E2 -26629.619} C_VEL
LIN {X 0,Y 99.583,Z 461.966,A -85,B 0,C 180,E1 -26636.965,E2 -26636.965} C_VEL
LIN {X 0,Y 99.908,Z 469.124,A -85,B 0,C 180,E1 -26644.033,E2 -26644.033} C_VEL
LIN {X 0,Y 101.32,Z 475.984,A -85,B 0,C 180,E1 -26652.01,E2 -26652.01} C_VEL
LIN {X 0,Y 105.074,Z 483.184,A -85,B 0,C 180,E1 -26661.584,E2 -26661.584} C_VEL
LIN {X 0,Y 113.07,Z 490.177,A -85,B 0,C 180,E1 -26671.892,E2 -26671.892} C_VEL
LIN {X 0,Y 125.274,Z 495.953,A -85,B 0,C 180,E1 -26681.155,E2 -26681.155} C_VEL
LIN {X 0,Y 124.218,Z 496.095,A -85,B 0,C 180,E1 -26682.646,E2 -26682.646} C_VEL
LIN {X 0,Y 112.845,Z 494.679,A -85,B 0,C 180,E1 -26691.476,E2 -26691.476} C_VEL
LIN {X 0,Y 105.196,Z 492.108,A -85,B 0,C 180,E1 -26702.115,E2 -26702.115} C_VEL
LIN {X 0,Y 101.952,Z 487.817,A -85,B 0,C 180,E1 -26714.812,E2 -26714.812} C_VEL
LIN {X 0,Y 102.621,Z 483.371,A -85,B 0,C 180,E1 -26724.101,E2 -26724.101} C_VEL
LIN {X 0,Y 103.027,Z 482.225,A -85,B 0,C 180,E1 -26726.086,E2 -26726.086} C_VEL
LIN {X 0,Y 103.121,Z 480.898,A -85,B 0,C 180,E1 -26728.045,E2 -26728.045} C_VEL
LIN {X 0,Y 102.76,Z 477.487,A -85,B 0,C 180,E1 -26731.957,E2 -26731.957} C_VEL
LIN {X 0,Y 102.211,Z 470.268,A -85,B 0,C 180,E1 -26738.897,E2 -26738.897} C_VEL
LIN {X 0,Y 102.497,Z 461.502,A -85,B 0,C 180,E1 -26745.916,E2 -26745.916} C_VEL
LIN {X 0,Y 103.91,Z 450.953,A -85,B 0,C 180,E1 -26752.884,E2 -26752.884} C_VEL
LIN {X 0,Y 106.668,Z 438.648,A -85,B 0,C 180,E1 -26759.561,E2 -26759.561} C_VEL
LIN {X 0,Y 110.341,Z 424.974,A -85,B 0,C 180,E1 -26765.532,E2 -26765.532} C_VEL
LIN {X 0,Y 114.637,Z 410.192,A -85,B 0,C 180,E1 -26770.643,E2 -26770.643} C_VEL
LIN {X 0,Y 119.318,Z 394.275,A -85,B 0,C 180,E1 -26774.973,E2 -26774.973} C_VEL
LIN {X 0,Y 123.605,Z 378.863,A -85,B 0,C 180,E1 -26778.265,E2 -26778.265} C_VEL
LIN {X 0,Y 128.275,Z 360.228,A -85,B 0,C 180,E1 -26781.324,E2 -26781.324} C_VEL
LIN {X 0,Y 132.038,Z 342.74,A -85,B 0,C 180,E1 -26783.483,E2 -26783.483} C_VEL
LIN {X 0,Y 136.384,Z 315.517,A -85,B 0,C 180,E1 -26786.026,E2 -26786.026} C_VEL
LIN {X 0,Y 139.047,Z 298.992,A -85,B 0,C 180,E1 -26787.403,E2 -26787.403} C_VEL
LIN {X 0,Y 139.352,Z 293.26,A -85,B 0,C 180,E1 -26788.004,E2 -26788.004} C_VEL
LIN {X 0,Y 137.503,Z 274.551,A -85,B 0,C 180,E1 -26790.636,E2 -26790.636} C_VEL
LIN {X 0,Y 138.063,Z 268.84,A -85,B 0,C 180,E1 -26791.19,E2 -26791.19} C_VEL
LIN {X 0,Y 142.56,Z 243.098,A -85,B 0,C 180,E1 -26793.148,E2 -26793.148} C_VEL
LIN {X 0,Y 134.776,Z 221.806,A -85,B 0,C 180,E1 -26798.075,E2 -26798.075} C_VEL
LIN {X 0,Y 128.528,Z 205.359,A -85,B 0,C 180,E1 -26802.531,E2 -26802.531} C_VEL
LIN {X 0,Y 124.858,Z 196.58,A -85,B 0,C 180,E1 -26805.328,E2 -26805.328} C_VEL
LIN {X 0,Y 117.909,Z 182.829,A -85,B 0,C 180,E1 -26810.821,E2 -26810.821} C_VEL
LIN {X 0,Y 111.674,Z 171.326,A -85,B 0,C 180,E1 -26816.518,E2 -26816.518} C_VEL
LIN {X 0,Y 106.251,Z 162.33,A -85,B 0,C 180,E1 -26822.27,E2 -26822.27} C_VEL
LIN {X 0,Y 104.96,Z 160.153,A -85,B 0,C 180,E1 -26823.84,E2 -26823.84} C_VEL
LIN {X 0,Y 102.45,Z 156.968,A -85,B 0,C 180,E1 -26826.831,E2 -26826.831} C_VEL
LIN {X 0,Y 101.658,Z 155.61,A -85,B 0,C 180,E1 -26827.948,E2 -26827.948} C_VEL
LIN {X 0,Y 99.201,Z 152.978,A -85,B 0,C 180,E1 -26831.233,E2 -26831.233} C_VEL
LIN {X 0,Y 98.059,Z 150.58,A -85,B 0,C 180,E1 -26833.275,E2 -26833.275} C_VEL
LIN {X 0,Y 95.256,Z 148.606,A -85,B 0,C 180,E1 -26837.58,E2 -26837.58} C_VEL
LIN {X 0,Y 93.973,Z 146.154,A -85,B 0,C 180,E1 -26840.522,E2 -26840.522} C_VEL
LIN {X 0,Y 93.71,Z 145.123,A -85,B 0,C 180,E1 -26841.446,E2 -26841.446} C_VEL
LIN {X 0,Y 93.62,Z 145.134,A -85,B 0,C 180,E1 -26846.771,E2 -26846.771} C_VEL
LIN {X 0,Y 93.59,Z 145.139,A -85,B 0,C 180,E1 -26854.312,E2 -26854.312} C_VEL
LIN {X 0,Y 93.536,Z 145.146,A -85,B 0,C 180,E1 -26862.55,E2 -26862.55} C_VEL
LIN {X 0,Y 93.554,Z 145.136,A -85,B 0,C 180,E1 -26868.697,E2 -26868.697} C_VEL
LIN {X 0,Y 93.601,Z 145.126,A -85,B 0,C 180,E1 -26875.684,E2 -26875.684} C_VEL
LIN {X 0,Y 93.668,Z 145.126,A -85,B 0,C 180,E1 -26884.207,E2 -26884.207} C_VEL
LIN {X 0,Y 93.795,Z 145.114,A -85,B 0,C 180,E1 -26891.858,E2 -26891.858} C_VEL
LIN {X 0,Y 94.701,Z 147.542,A -85,B 0,C 180,E1 -26894.402,E2 -26894.402} C_VEL
LIN {X 0,Y 97.473,Z 150.231,A -85,B 0,C 180,E1 -26899.093,E2 -26899.093} C_VEL
LIN {X 0,Y 98.337,Z 150.931,A -85,B 0,C 180,E1 -26900.36,E2 -26900.36} C_VEL
LIN {X 0,Y 100.004,Z 154.016,A -85,B 0,C 180,E1 -26903.122,E2 -26903.122} C_VEL
LIN {X 0,Y 102.502,Z 156.348,A -85,B 0,C 180,E1 -26906.225,E2 -26906.225} C_VEL
LIN {X 0,Y 105.129,Z 160.709,A -85,B 0,C 180,E1 -26909.588,E2 -26909.588} C_VEL
LIN {X 0,Y 108.665,Z 166.588,A -85,B 0,C 180,E1 -26913.595,E2 -26913.595} C_VEL
LIN {X 0,Y 111.653,Z 171.534,A -85,B 0,C 180,E1 -26916.614,E2 -26916.614} C_VEL
LIN {X 0,Y 117.855,Z 183.102,A -85,B 0,C 180,E1 -26922.278,E2 -26922.278} C_VEL
LIN {X 0,Y 123.751,Z 194.756,A -85,B 0,C 180,E1 -26926.957,E2 -26926.957} C_VEL
LIN {X 0,Y 131.406,Z 211.156,A -85,B 0,C 180,E1 -26932.313,E2 -26932.313} C_VEL
LIN {X 0,Y 139.172,Z 229.169,A -85,B 0,C 180,E1 -26937.136,E2 -26937.136} C_VEL
LIN {X 0,Y 140.564,Z 232.6,A -85,B 0,C 180,E1 -26937.954,E2 -26937.954} C_VEL
LIN {X 0,Y 125.657,Z 320.772,A -85,B 0,C 180,E1 -26945.291,E2 -26945.291} C_VEL
LIN {X 0,Y 121.961,Z 339.363,A -85,B 0,C 180,E1 -26947.594,E2 -26947.594} C_VEL
LIN {X 0,Y 117.785,Z 357.068,A -85,B 0,C 180,E1 -26950.485,E2 -26950.485} C_VEL
LIN {X 0,Y 113.33,Z 373.371,A -85,B 0,C 180,E1 -26953.87,E2 -26953.87} C_VEL
LIN {X 0,Y 108.407,Z 390.239,A -85,B 0,C 180,E1 -26958.355,E2 -26958.355} C_VEL
LIN {X 0,Y 103.76,Z 405.797,A -85,B 0,C 180,E1 -26963.654,E2 -26963.654} C_VEL
LIN {X 0,Y 99.368,Z 421.192,A -85,B 0,C 180,E1 -26970.324,E2 -26970.324} C_VEL
LIN {X 0,Y 96.029,Z 434.206,A -85,B 0,C 180,E1 -26977.404,E2 -26977.404} C_VEL
LIN {X 0,Y 93.878,Z 445.307,A -85,B 0,C 180,E1 -26984.81,E2 -26984.81} C_VEL
LIN {X 0,Y 92.892,Z 454.872,A -85,B 0,C 180,E1 -26992.391,E2 -26992.391} C_VEL
LIN {X 0,Y 92.812,Z 464.102,A -85,B 0,C 180,E1 -27001.084,E2 -27001.084} C_VEL
LIN {X 0,Y 93.704,Z 470.856,A -85,B 0,C 180,E1 -27008.627,E2 -27008.627} C_VEL
LIN {X 0,Y 95.84,Z 477.435,A -85,B 0,C 180,E1 -27017.056,E2 -27017.056} C_VEL
LIN {X 0,Y 101.1,Z 484.408,A -85,B 0,C 180,E1 -27026.862,E2 -27026.862} C_VEL
LIN {X 0,Y 110.796,Z 491.236,A -85,B 0,C 180,E1 -27037.056,E2 -27037.056} C_VEL
LIN {X 0,Y 116.781,Z 494.058,A -85,B 0,C 180,E1 -27041.451,E2 -27041.451} C_VEL
LIN {X 0,Y 115.212,Z 493.969,A -85,B 0,C 180,E1 -27042.942,E2 -27042.942} C_VEL
LIN {X 0,Y 104.26,Z 491.893,A -85,B 0,C 180,E1 -27052.647,E2 -27052.647} C_VEL
LIN {X 0,Y 97.462,Z 488.615,A -85,B 0,C 180,E1 -27064.361,E2 -27064.361} C_VEL
LIN {X 0,Y 95.42,Z 483.853,A -85,B 0,C 180,E1 -27077.232,E2 -27077.232} C_VEL
LIN {X 0,Y 96.466,Z 479.511,A -85,B 0,C 180,E1 -27085.819,E2 -27085.819} C_VEL
LIN {X 0,Y 96.522,Z 478.015,A -85,B 0,C 180,E1 -27087.911,E2 -27087.911} C_VEL
LIN {X 0,Y 96.002,Z 474.427,A -85,B 0,C 180,E1 -27092.095,E2 -27092.095} C_VEL
LIN {X 0,Y 95.503,Z 468.027,A -85,B 0,C 180,E1 -27098.461,E2 -27098.461} C_VEL
LIN {X 0,Y 95.724,Z 459.048,A -85,B 0,C 180,E1 -27105.974,E2 -27105.974} C_VEL
LIN {X 0,Y 97.187,Z 448.303,A -85,B 0,C 180,E1 -27113.433,E2 -27113.433} C_VEL
LIN {X 0,Y 100.099,Z 435.726,A -85,B 0,C 180,E1 -27120.564,E2 -27120.564} C_VEL
LIN {X 0,Y 103.994,Z 421.734,A -85,B 0,C 180,E1 -27126.85,E2 -27126.85} C_VEL
LIN {X 0,Y 108.558,Z 406.624,A -85,B 0,C 180,E1 -27132.193,E2 -27132.193} C_VEL
LIN {X 0,Y 113.47,Z 390.295,A -85,B 0,C 180,E1 -27136.668,E2 -27136.668} C_VEL
LIN {X 0,Y 118.21,Z 373.315,A -85,B 0,C 180,E1 -27140.243,E2 -27140.243} C_VEL
LIN {X 0,Y 122.874,Z 354.705,A -85,B 0,C 180,E1 -27143.198,E2 -27143.198} C_VEL
LIN {X 0,Y 126.393,Z 337.548,A -85,B 0,C 180,E1 -27145.272,E2 -27145.272} C_VEL
LIN {X 0,Y 138.063,Z 268.84,A -85,B 0,C 180,E1 -27151.19,E2 -27151.19} C_VEL
LIN {X 0,Y 138.766,Z 263.09,A -85,B 0,C 180,E1 -27151.716,E2 -27151.716} C_VEL
LIN {X 0,Y 138.624,Z 257.41,A -85,B 0,C 180,E1 -27152.446,E2 -27152.446} C_VEL
LIN {X 0,Y 137.463,Z 250.054,A -85,B 0,C 180,E1 -27153.661,E2 -27153.661} C_VEL
LIN {X 0,Y 134.482,Z 239.526,A -85,B 0,C 180,E1 -27155.844,E2 -27155.844} C_VEL
LIN {X 0,Y 127.587,Z 220.393,A -85,B 0,C 180,E1 -27160.701,E2 -27160.701} C_VEL
LIN {X 0,Y 121.125,Z 203.195,A -85,B 0,C 180,E1 -27165.854,E2 -27165.854} C_VEL
LIN {X 0,Y 114.761,Z 190.085,A -85,B 0,C 180,E1 -27171.141,E2 -27171.141} C_VEL
LIN {X 0,Y 107.846,Z 176.703,A -85,B 0,C 180,E1 -27177.872,E2 -27177.872} C_VEL
LIN {X 0,Y 101.928,Z 166.296,A -85,B 0,C 180,E1 -27184.817,E2 -27184.817} C_VEL
LIN {X 0,Y 99.366,Z 163.006,A -85,B 0,C 180,E1 -27188.048,E2 -27188.048} C_VEL
LIN {X 0,Y 98.466,Z 161.636,A -85,B 0,C 180,E1 -27189.37,E2 -27189.37} C_VEL
LIN {X 0,Y 96.134,Z 158.814,A -85,B 0,C 180,E1 -27192.779,E2 -27192.779} C_VEL
LIN {X 0,Y 95.235,Z 157.036,A -85,B 0,C 180,E1 -27194.502,E2 -27194.502} C_VEL
LIN {X 0,Y 92.444,Z 154.618,A -85,B 0,C 180,E1 -27199.285,E2 -27199.285} C_VEL
LIN {X 0,Y 91.195,Z 151.764,A -85,B 0,C 180,E1 -27202.665,E2 -27202.665} C_VEL
LIN {X 0,Y 88.069,Z 149.608,A -85,B 0,C 180,E1 -27210.91,E2 -27210.91} C_VEL
LIN {X 0,Y 86.453,Z 146.034,A -85,B 0,C 180,E1 -27223.162,E2 -27223.162} C_VEL
LIN {X 0,Y 86.458,Z 146.03,A -85,B 0,C 180,E1 -27230.119,E2 -27230.119} C_VEL
LIN {X 0,Y 87.186,Z 148.176,A -85,B 0,C 180,E1 -27238.066,E2 -27238.066} C_VEL
LIN {X 0,Y 89.847,Z 151.09,A -85,B 0,C 180,E1 -27247.587,E2 -27247.587} C_VEL
LIN {X 0,Y 91.323,Z 151.998,A -85,B 0,C 180,E1 -27250.911,E2 -27250.911} C_VEL
LIN {X 0,Y 93.044,Z 155.07,A -85,B 0,C 180,E1 -27255.023,E2 -27255.023} C_VEL
LIN {X 0,Y 95.512,Z 157.305,A -85,B 0,C 180,E1 -27259.134,E2 -27259.134} C_VEL
LIN {X 0,Y 97.526,Z 160.673,A -85,B 0,C 180,E1 -27262.56,E2 -27262.56} C_VEL
LIN {X 0,Y 99.569,Z 162.7,A -85,B 0,C 180,E1 -27265.223,E2 -27265.223} C_VEL
LIN {X 0,Y 101.603,Z 166.241,A -85,B 0,C 180,E1 -27268.051,E2 -27268.051} C_VEL
LIN {X 0,Y 106.616,Z 174.77,A -85,B 0,C 180,E1 -27273.973,E2 -27273.973} C_VEL
LIN {X 0,Y 112.688,Z 186.233,A -85,B 0,C 180,E1 -27280.094,E2 -27280.094} C_VEL
LIN {X 0,Y 118.903,Z 198.856,A -85,B 0,C 180,E1 -27285.478,E2 -27285.478} C_VEL
LIN {X 0,Y 126.712,Z 216.133,A -85,B 0,C 180,E1 -27291.357,E2 -27291.357} C_VEL
LIN {X 0,Y 134.341,Z 234.44,A -85,B 0,C 180,E1 -27296.39,E2 -27296.39} C_VEL
LIN {X 0,Y 125.806,Z 282.744,A -85,B 0,C 180,E1 -27300.301,E2 -27300.301} C_VEL
LIN {X 0,Y 118.831,Z 322.962,A -85,B 0,C 180,E1 -27304.105,E2 -27304.105} C_VEL
LIN {X 0,Y 115.167,Z 340.47,A -85,B 0,C 180,E1 -27306.412,E2 -27306.412} C_VEL
LIN {X 0,Y 110.581,Z 358.953,A -85,B 0,C 180,E1 -27309.614,E2 -27309.614} C_VEL
LIN {X 0,Y 105.529,Z 376.502,A -85,B 0,C 180,E1 -27313.593,E2 -27313.593} C_VEL
LIN {X 0,Y 100.569,Z 392.866,A -85,B 0,C 180,E1 -27318.403,E2 -27318.403} C_VEL
LIN {X 0,Y 96.217,Z 406.95,A -85,B 0,C 180,E1 -27323.643,E2 -27323.643} C_VEL
LIN {X 0,Y 92.117,Z 421.093,A -85,B 0,C 180,E1 -27330.27,E2 -27330.27} C_VEL
LIN {X 0,Y 88.805,Z 434.105,A -85,B 0,C 180,E1 -27337.919,E2 -27337.919} C_VEL
LIN {X 0,Y 86.594,Z 446.432,A -85,B 0,C 180,E1 -27346.899,E2 -27346.899} C_VEL
LIN {X 0,Y 85.888,Z 455.973,A -85,B 0,C 180,E1 -27355.306,E2 -27355.306} C_VEL
LIN {X 0,Y 86.163,Z 463.904,A -85,B 0,C 180,E1 -27363.507,E2 -27363.507} C_VEL
LIN {X 0,Y 87.427,Z 470.689,A -85,B 0,C 180,E1 -27371.593,E2 -27371.593} C_VEL
LIN {X 0,Y 91.226,Z 478.75,A -85,B 0,C 180,E1 -27382.655,E2 -27382.655} C_VEL
LIN {X 0,Y 97.98,Z 485.517,A -85,B 0,C 180,E1 -27392.545,E2 -27392.545} C_VEL
LIN {X 0,Y 107.336,Z 491.17,A -85,B 0,C 180,E1 -27400.901,E2 -27400.901} C_VEL
LIN {X 0,Y 107.453,Z 491.582,A -85,B 0,C 180,E1 -27402.502,E2 -27402.502} C_VEL
LIN {X 0,Y 95.912,Z 488.663,A -85,B 0,C 180,E1 -27414.109,E2 -27414.109} C_VEL
LIN {X 0,Y 90.052,Z 484.655,A -85,B 0,C 180,E1 -27427.029,E2 -27427.029} C_VEL
LIN {X 0,Y 89.086,Z 480.103,A -85,B 0,C 180,E1 -27438.622,E2 -27438.622} C_VEL
LIN {X 0,Y 89.992,Z 476.615,A -85,B 0,C 180,E1 -27445.518,E2 -27445.518} C_VEL
LIN {X 0,Y 89.885,Z 475.064,A -85,B 0,C 180,E1 -27447.757,E2 -27447.757} C_VEL
LIN {X 0,Y 89.071,Z 469.122,A -85,B 0,C 180,E1 -27454.522,E2 -27454.522} C_VEL
LIN {X 0,Y 88.75,Z 460.68,A -85,B 0,C 180,E1 -27462.575,E2 -27462.575} C_VEL
LIN {X 0,Y 89.668,Z 450.417,A -85,B 0,C 180,E1 -27470.647,E2 -27470.647} C_VEL
LIN {X 0,Y 92.139,Z 438.369,A -85,B 0,C 180,E1 -27478.468,E2 -27478.468} C_VEL
LIN {X 0,Y 95.704,Z 425.143,A -85,B 0,C 180,E1 -27485.319,E2 -27485.319} C_VEL
LIN {X 0,Y 100.483,Z 409.547,A -85,B 0,C 180,E1 -27491.636,E2 -27491.636} C_VEL
LIN {X 0,Y 105.325,Z 393.802,A -85,B 0,C 180,E1 -27496.519,E2 -27496.519} C_VEL
LIN {X 0,Y 110.267,Z 377.252,A -85,B 0,C 180,E1 -27500.465,E2 -27500.465} C_VEL
LIN {X 0,Y 115.013,Z 359.516,A -85,B 0,C 180,E1 -27503.687,E2 -27503.687} C_VEL
LIN {X 0,Y 119.091,Z 341.772,A -85,B 0,C 180,E1 -27506.082,E2 -27506.082} C_VEL
LIN {X 0,Y 123.819,Z 314.207,A -85,B 0,C 180,E1 -27508.871,E2 -27508.871} C_VEL
LIN {X 0,Y 136.34,Z 244.904,A -85,B 0,C 180,E1 -27514.604,E2 -27514.604} C_VEL
LIN {X 0,Y 134.482,Z 239.526,A -85,B 0,C 180,E1 -27515.844,E2 -27515.844} C_VEL
LIN {X 0,Y 132.276,Z 234.93,A -85,B 0,C 180,E1 -27517.12,E2 -27517.12} C_VEL
LIN {X 0,Y 127.247,Z 228.577,A -85,B 0,C 180,E1 -27519.652,E2 -27519.652} C_VEL
LIN {X 0,Y 122.271,Z 222.311,A -85,B 0,C 180,E1 -27522.395,E2 -27522.395} C_VEL
LIN {X 0,Y 120.124,Z 217.832,A -85,B 0,C 180,E1 -27523.937,E2 -27523.937} C_VEL
LIN {X 0,Y 115.661,Z 205.987,A -85,B 0,C 180,E1 -27527.862,E2 -27527.862} C_VEL
LIN {X 0,Y 109.235,Z 192.465,A -85,B 0,C 180,E1 -27533.749,E2 -27533.749} C_VEL
LIN {X 0,Y 103.71,Z 181.562,A -85,B 0,C 180,E1 -27539.66,E2 -27539.66} C_VEL
LIN {X 0,Y 98.629,Z 172.243,A -85,B 0,C 180,E1 -27546.125,E2 -27546.125} C_VEL
LIN {X 0,Y 95.944,Z 168.366,A -85,B 0,C 180,E1 -27549.919,E2 -27549.919} C_VEL
LIN {X 0,Y 93.03,Z 164.442,A -85,B 0,C 180,E1 -27554.641,E2 -27554.641} C_VEL
LIN {X 0,Y 92.399,Z 163.353,A -85,B 0,C 180,E1 -27555.847,E2 -27555.847} C_VEL
LIN {X 0,Y 89.84,Z 160.754,A -85,B 0,C 180,E1 -27560.783,E2 -27560.783} C_VEL
LIN {X 0,Y 88.727,Z 158.39,A -85,B 0,C 180,E1 -27563.902,E2 -27563.902} C_VEL
LIN {X 0,Y 85.703,Z 155.781,A -85,B 0,C 180,E1 -27573.365,E2 -27573.365} C_VEL
LIN {X 0,Y 84.685,Z 152.911,A -85,B 0,C 180,E1 -27583.211,E2 -27583.211} C_VEL
LIN {X 0,Y 84.667,Z 152.922,A -85,B 0,C 180,E1 -27589.808,E2 -27589.808} C_VEL
LIN {X 0,Y 85.289,Z 155.03,A -85,B 0,C 180,E1 -27597.616,E2 -27597.616} C_VEL
LIN {X 0,Y 88.373,Z 158.164,A -85,B 0,C 180,E1 -27608.474,E2 -27608.474} C_VEL
LIN {X 0,Y 88.981,Z 158.705,A -85,B 0,C 180,E1 -27609.962,E2 -27609.962} C_VEL
LIN {X 0,Y 90.775,Z 161.728,A -85,B 0,C 180,E1 -27614.371,E2 -27614.371} C_VEL
LIN {X 0,Y 92.82,Z 163.826,A -85,B 0,C 180,E1 -27618.076,E2 -27618.076} C_VEL
LIN {X 0,Y 94.881,Z 167.101,A -85,B 0,C 180,E1 -27621.701,E2 -27621.701} C_VEL
LIN {X 0,Y 96.646,Z 168.979,A -85,B 0,C 180,E1 -27624.158,E2 -27624.158} C_VEL
LIN {X 0,Y 98.835,Z 173.182,A -85,B 0,C 180,E1 -27627.459,E2 -27627.459} C_VEL
LIN {X 0,Y 102.692,Z 179.819,A -85,B 0,C 180,E1 -27632.299,E2 -27632.299} C_VEL
LIN {X 0,Y 108.579,Z 191.486,A -85,B 0,C 180,E1 -27638.777,E2 -27638.777} C_VEL
LIN {X 0,Y 114.426,Z 203.807,A -85,B 0,C 180,E1 -27644.224,E2 -27644.224} C_VEL
LIN {X 0,Y 121.057,Z 218.851,A -85,B 0,C 180,E1 -27649.613,E2 -27649.613} C_VEL
LIN {X 0,Y 128.187,Z 236.287,A -85,B 0,C 180,E1 -27654.715,E2 -27654.715} C_VEL
LIN {X 0,Y 124.099,Z 258.817,A -85,B 0,C 180,E1 -27656.562,E2 -27656.562} C_VEL
LIN {X 0,Y 112.653,Z 321.961,A -85,B 0,C 180,E1 -27662.417,E2 -27662.417} C_VEL
LIN {X 0,Y 108.716,Z 340.211,A -85,B 0,C 180,E1 -27664.898,E2 -27664.898} C_VEL
LIN {X 0,Y 103.982,Z 358.609,A -85,B 0,C 180,E1 -27668.213,E2 -27668.213} C_VEL
LIN {X 0,Y 99.241,Z 374.727,A -85,B 0,C 180,E1 -27671.962,E2 -27671.962} C_VEL
LIN {X 0,Y 94.023,Z 391.284,A -85,B 0,C 180,E1 -27676.994,E2 -27676.994} C_VEL
LIN {X 0,Y 89.057,Z 406.93,A -85,B 0,C 180,E1 -27683.155,E2 -27683.155} C_VEL
LIN {X 0,Y 84.897,Z 420.871,A -85,B 0,C 180,E1 -27690.218,E2 -27690.218} C_VEL
LIN {X 0,Y 81.595,Z 433.887,A -85,B 0,C 180,E1 -27698.526,E2 -27698.526} C_VEL
LIN {X 0,Y 79.599,Z 445.72,A -85,B 0,C 180,E1 -27707.886,E2 -27707.886} C_VEL
LIN {X 0,Y 79.052,Z 454.535,A -85,B 0,C 180,E1 -27716.176,E2 -27716.176} C_VEL
LIN {X 0,Y 79.512,Z 462.548,A -85,B 0,C 180,E1 -27725.07,E2 -27725.07} C_VEL
LIN {X 0,Y 80.78,Z 468.511,A -85,B 0,C 180,E1 -27732.562,E2 -27732.562} C_VEL
LIN {X 0,Y 84.99,Z 477.027,A -85,B 0,C 180,E1 -27744.54,E2 -27744.54} C_VEL
LIN {X 0,Y 93.994,Z 485.318,A -85,B 0,C 180,E1 -27756.738,E2 -27756.738} C_VEL
LIN {X 0,Y 99.088,Z 488.363,A -85,B 0,C 180,E1 -27761.162,E2 -27761.162} C_VEL
LIN {X 0,Y 98.868,Z 488.625,A -85,B 0,C 180,E1 -27762.809,E2 -27762.809} C_VEL
LIN {X 0,Y 90.514,Z 486.203,A -85,B 0,C 180,E1 -27771.595,E2 -27771.595} C_VEL
LIN {X 0,Y 83.955,Z 481.994,A -85,B 0,C 180,E1 -27785.253,E2 -27785.253} C_VEL
LIN {X 0,Y 82.713,Z 477.229,A -85,B 0,C 180,E1 -27797.733,E2 -27797.733} C_VEL
LIN {X 0,Y 83.519,Z 473.607,A -85,B 0,C 180,E1 -27805.17,E2 -27805.17} C_VEL
LIN {X 0,Y 82.93,Z 469.97,A -85,B 0,C 180,E1 -27809.997,E2 -27809.997} C_VEL
LIN {X 0,Y 82.15,Z 463.257,A -85,B 0,C 180,E1 -27817.37,E2 -27817.37} C_VEL
LIN {X 0,Y 82.23,Z 453.841,A -85,B 0,C 180,E1 -27826.124,E2 -27826.124} C_VEL
LIN {X 0,Y 83.909,Z 442.602,A -85,B 0,C 180,E1 -27834.754,E2 -27834.754} C_VEL
LIN {X 0,Y 86.924,Z 430.311,A -85,B 0,C 180,E1 -27842.384,E2 -27842.384} C_VEL
LIN {X 0,Y 90.932,Z 416.769,A -85,B 0,C 180,E1 -27849.071,E2 -27849.071} C_VEL
LIN {X 0,Y 95.816,Z 401.473,A -85,B 0,C 180,E1 -27854.905,E2 -27854.905} C_VEL
LIN {X 0,Y 101.187,Z 384.543,A -85,B 0,C 180,E1 -27859.815,E2 -27859.815} C_VEL
LIN {X 0,Y 105.932,Z 368.242,A -85,B 0,C 180,E1 -27863.398,E2 -27863.398} C_VEL
LIN {X 0,Y 110.728,Z 349.866,A -85,B 0,C 180,E1 -27866.409,E2 -27866.409} C_VEL
LIN {X 0,Y 114.14,Z 333.355,A -85,B 0,C 180,E1 -27868.47,E2 -27868.47} C_VEL
LIN {X 0,Y 130.112,Z 246.806,A -85,B 0,C 180,E1 -27876.172,E2 -27876.172} C_VEL
LIN {X 0,Y 125.167,Z 232.061,A -85,B 0,C 180,E1 -27879.858,E2 -27879.858} C_VEL
LIN {X 0,Y 120.124,Z 217.832,A -85,B 0,C 180,E1 -27883.937,E2 -27883.937} C_VEL
LIN {X 0,Y 118,Z 213.452,A -85,B 0,C 180,E1 -27885.529,E2 -27885.529} C_VEL
LIN {X 0,Y 115.214,Z 209.85,A -85,B 0,C 180,E1 -27887.4,E2 -27887.4} C_VEL
LIN {X 0,Y 107.226,Z 201.355,A -85,B 0,C 180,E1 -27893.12,E2 -27893.12} C_VEL
LIN {X 0,Y 105.643,Z 198.828,A -85,B 0,C 180,E1 -27894.576,E2 -27894.576} C_VEL
LIN {X 0,Y 100.015,Z 187.036,A -85,B 0,C 180,E1 -27901.127,E2 -27901.127} C_VEL
LIN {X 0,Y 95.264,Z 177.997,A -85,B 0,C 180,E1 -27907.709,E2 -27907.709} C_VEL
LIN {X 0,Y 92.312,Z 173.678,A -85,B 0,C 180,E1 -27912.237,E2 -27912.237} C_VEL
LIN {X 0,Y 89.996,Z 170.105,A -85,B 0,C 180,E1 -27916.518,E2 -27916.518} C_VEL
LIN {X 0,Y 87.041,Z 166.581,A -85,B 0,C 180,E1 -27922.866,E2 -27922.866} C_VEL
LIN {X 0,Y 86.321,Z 164.948,A -85,B 0,C 180,E1 -27925.205,E2 -27925.205} C_VEL
LIN {X 0,Y 83.61,Z 162.302,A -85,B 0,C 180,E1 -27934.743,E2 -27934.743} C_VEL
LIN {X 0,Y 82.889,Z 159.779,A -85,B 0,C 180,E1 -27943.545,E2 -27943.545} C_VEL
LIN {X 0,Y 82.892,Z 159.999,A -85,B 0,C 180,E1 -27950.515,E2 -27950.515} C_VEL
LIN {X 0,Y 83.425,Z 161.993,A -85,B 0,C 180,E1 -27957.398,E2 -27957.398} C_VEL
LIN {X 0,Y 86.641,Z 165.308,A -85,B 0,C 180,E1 -27968.865,E2 -27968.865} C_VEL
LIN {X 0,Y 88.663,Z 168.527,A -85,B 0,C 180,E1 -27973.988,E2 -27973.988} C_VEL
LIN {X 0,Y 90.139,Z 170.243,A -85,B 0,C 180,E1 -27976.913,E2 -27976.913} C_VEL
LIN {X 0,Y 92.471,Z 173.751,A -85,B 0,C 180,E1 -27981.128,E2 -27981.128} C_VEL
LIN {X 0,Y 93.753,Z 175.317,A -85,B 0,C 180,E1 -27983.088,E2 -27983.088} C_VEL
LIN {X 0,Y 98.925,Z 185.122,A -85,B 0,C 180,E1 -27990.665,E2 -27990.665} C_VEL
LIN {X 0,Y 104.375,Z 196.392,A -85,B 0,C 180,E1 -27997.197,E2 -27997.197} C_VEL
LIN {X 0,Y 109.8,Z 208.312,A -85,B 0,C 180,E1 -28002.705,E2 -28002.705} C_VEL
LIN {X 0,Y 116.553,Z 224.26,A -85,B 0,C 180,E1 -28008.646,E2 -28008.646} C_VEL
LIN {X 0,Y 122.172,Z 238.558,A -85,B 0,C 180,E1 -28013.014,E2 -28013.014} C_VEL
LIN {X 0,Y 106.163,Z 322.894,A -85,B 0,C 180,E1 -28020.847,E2 -28020.847} C_VEL
LIN {X 0,Y 102.367,Z 339.762,A -85,B 0,C 180,E1 -28023.206,E2 -28023.206} C_VEL
LIN {X 0,Y 97.417,Z 358.278,A -85,B 0,C 180,E1 -28026.667,E2 -28026.667} C_VEL
LIN {X 0,Y 92.001,Z 375.891,A -85,B 0,C 180,E1 -28031.03,E2 -28031.03} C_VEL
LIN {X 0,Y 87.12,Z 390.952,A -85,B 0,C 180,E1 -28035.913,E2 -28035.913} C_VEL
LIN {X 0,Y 82.014,Z 406.394,A -85,B 0,C 180,E1 -28042.428,E2 -28042.428} C_VEL
LIN {X 0,Y 78.019,Z 419.508,A -85,B 0,C 180,E1 -28049.555,E2 -28049.555} C_VEL
LIN {X 0,Y 74.798,Z 431.813,A -85,B 0,C 180,E1 -28057.923,E2 -28057.923} C_VEL
LIN {X 0,Y 72.787,Z 443.205,A -85,B 0,C 180,E1 -28067.451,E2 -28067.451} C_VEL
LIN {X 0,Y 72.306,Z 452.891,A -85,B 0,C 180,E1 -28077.214,E2 -28077.214} C_VEL
LIN {X 0,Y 72.951,Z 461.137,A -85,B 0,C 180,E1 -28086.916,E2 -28086.916} C_VEL
LIN {X 0,Y 74.892,Z 468.103,A -85,B 0,C 180,E1 -28096.351,E2 -28096.351} C_VEL
LIN {X 0,Y 80.105,Z 476.547,A -85,B 0,C 180,E1 -28108.848,E2 -28108.848} C_VEL
LIN {X 0,Y 90.418,Z 484.819,A -85,B 0,C 180,E1 -28121.056,E2 -28121.056} C_VEL
LIN {X 0,Y 91.514,Z 485.501,A -85,B 0,C 180,E1 -28121.977,E2 -28121.977} C_VEL
LIN {X 0,Y 85.358,Z 483.64,A -85,B 0,C 180,E1 -28128.797,E2 -28128.797} C_VEL
LIN {X 0,Y 78.043,Z 479.122,A -85,B 0,C 180,E1 -28143.235,E2 -28143.235} C_VEL
LIN {X 0,Y 76.423,Z 474.221,A -85,B 0,C 180,E1 -28156.705,E2 -28156.705} C_VEL
LIN {X 0,Y 76.854,Z 471.811,A -85,B 0,C 180,E1 -28162.112,E2 -28162.112} C_VEL
LIN {X 0,Y 77.064,Z 470.399,A -85,B 0,C 180,E1 -28164.764,E2 -28164.764} C_VEL
LIN {X 0,Y 76.119,Z 465.418,A -85,B 0,C 180,E1 -28171.319,E2 -28171.319} C_VEL
LIN {X 0,Y 75.378,Z 456.77,A -85,B 0,C 180,E1 -28180.743,E2 -28180.743} C_VEL
LIN {X 0,Y 76.017,Z 446.464,A -85,B 0,C 180,E1 -28190.169,E2 -28190.169} C_VEL
LIN {X 0,Y 78.626,Z 434.019,A -85,B 0,C 180,E1 -28199.443,E2 -28199.443} C_VEL
LIN {X 0,Y 82.49,Z 420.445,A -85,B 0,C 180,E1 -28207.366,E2 -28207.366} C_VEL
LIN {X 0,Y 87.662,Z 404.586,A -85,B 0,C 180,E1 -28214.413,E2 -28214.413} C_VEL
LIN {X 0,Y 93.046,Z 388.145,A -85,B 0,C 180,E1 -28219.881,E2 -28219.881} C_VEL
LIN {X 0,Y 98.513,Z 370.464,A -85,B 0,C 180,E1 -28224.22,E2 -28224.22} C_VEL
LIN {X 0,Y 103.369,Z 352.904,A -85,B 0,C 180,E1 -28227.415,E2 -28227.415} C_VEL
LIN {X 0,Y 107.115,Z 336.596,A -85,B 0,C 180,E1 -28229.673,E2 -28229.673} C_VEL
LIN {X 0,Y 123.994,Z 248.034,A -85,B 0,C 180,E1 -28237.944,E2 -28237.944} C_VEL
LIN {X 0,Y 116.938,Z 227.214,A -85,B 0,C 180,E1 -28243.727,E2 -28243.727} C_VEL
LIN {X 0,Y 111.265,Z 211.051,A -85,B 0,C 180,E1 -28249.077,E2 -28249.077} C_VEL
LIN {X 0,Y 105.643,Z 198.828,A -85,B 0,C 180,E1 -28254.576,E2 -28254.576} C_VEL
LIN {X 0,Y 103.915,Z 196.673,A -85,B 0,C 180,E1 -28256.142,E2 -28256.142} C_VEL
LIN {X 0,Y 100.258,Z 194.602,A -85,B 0,C 180,E1 -28259.103,E2 -28259.103} C_VEL
LIN {X 0,Y 96.83,Z 192.556,A -85,B 0,C 180,E1 -28262.28,E2 -28262.28} C_VEL
LIN {X 0,Y 95.342,Z 190.433,A -85,B 0,C 180,E1 -28264.09,E2 -28264.09} C_VEL
LIN {X 0,Y 91.985,Z 183.761,A -85,B 0,C 180,E1 -28269.296,E2 -28269.296} C_VEL
LIN {X 0,Y 89.312,Z 179.664,A -85,B 0,C 180,E1 -28273.828,E2 -28273.828} C_VEL
LIN {X 0,Y 86.958,Z 175.995,A -85,B 0,C 180,E1 -28278.595,E2 -28278.595} C_VEL
LIN {X 0,Y 84.524,Z 172.712,A -85,B 0,C 180,E1 -28284.566,E2 -28284.566} C_VEL
LIN {X 0,Y 84.021,Z 171.531,A -85,B 0,C 180,E1 -28286.409,E2 -28286.409} C_VEL
LIN {X 0,Y 81.526,Z 168.76,A -85,B 0,C 180,E1 -28296.438,E2 -28296.438} C_VEL
LIN {X 0,Y 81.087,Z 166.681,A -85,B 0,C 180,E1 -28303.899,E2 -28303.899} C_VEL
LIN {X 0,Y 81.098,Z 166.878,A -85,B 0,C 180,E1 -28310.276,E2 -28310.276} C_VEL
LIN {X 0,Y 83.709,Z 171.325,A -85,B 0,C 180,E1 -28325.971,E2 -28325.971} C_VEL
LIN {X 0,Y 84.43,Z 172.046,A -85,B 0,C 180,E1 -28328.005,E2 -28328.005} C_VEL
LIN {X 0,Y 86.355,Z 175.139,A -85,B 0,C 180,E1 -28333.227,E2 -28333.227} C_VEL
LIN {X 0,Y 87.403,Z 176.428,A -85,B 0,C 180,E1 -28335.445,E2 -28335.445} C_VEL
LIN {X 0,Y 89.823,Z 180.145,A -85,B 0,C 180,E1 -28340.148,E2 -28340.148} C_VEL
LIN {X 0,Y 90.887,Z 181.663,A -85,B 0,C 180,E1 -28341.954,E2 -28341.954} C_VEL
LIN {X 0,Y 95.488,Z 191.03,A -85,B 0,C 180,E1 -28349.349,E2 -28349.349} C_VEL
LIN {X 0,Y 100.633,Z 202.315,A -85,B 0,C 180,E1 -28356.058,E2 -28356.058} C_VEL
LIN {X 0,Y 105.363,Z 213.163,A -85,B 0,C 180,E1 -28361.26,E2 -28361.26} C_VEL
LIN {X 0,Y 111.55,Z 228.38,A -85,B 0,C 180,E1 -28367.18,E2 -28367.18} C_VEL
LIN {X 0,Y 116.179,Z 240.302,A -85,B 0,C 180,E1 -28371.081,E2 -28371.081} C_VEL
LIN {X 0,Y 99.815,Z 323.172,A -85,B 0,C 180,E1 -28379.022,E2 -28379.022} C_VEL
LIN {X 0,Y 95.669,Z 340.674,A -85,B 0,C 180,E1 -28381.577,E2 -28381.577} C_VEL
LIN {X 0,Y 91.011,Z 357.554,A -85,B 0,C 180,E1 -28384.867,E2 -28384.867} C_VEL
LIN {X 0,Y 85.346,Z 375.337,A -85,B 0,C 180,E1 -28389.465,E2 -28389.465} C_VEL
LIN {X 0,Y 79.792,Z 391.833,A -85,B 0,C 180,E1 -28395.2,E2 -28395.2} C_VEL
LIN {X 0,Y 74.59,Z 406.993,A -85,B 0,C 180,E1 -28402.233,E2 -28402.233} C_VEL
LIN {X 0,Y 70.835,Z 419.051,A -85,B 0,C 180,E1 -28409.437,E2 -28409.437} C_VEL
LIN {X 0,Y 67.64,Z 431.39,A -85,B 0,C 180,E1 -28418.677,E2 -28418.677} C_VEL
LIN {X 0,Y 65.809,Z 442.785,A -85,B 0,C 180,E1 -28429.228,E2 -28429.228} C_VEL
LIN {X 0,Y 65.598,Z 451.176,A -85,B 0,C 180,E1 -28438.465,E2 -28438.465} C_VEL
LIN {X 0,Y 66.341,Z 458.397,A -85,B 0,C 180,E1 -28447.609,E2 -28447.609} C_VEL
LIN {X 0,Y 68.49,Z 465.675,A -85,B 0,C 180,E1 -28457.928,E2 -28457.928} C_VEL
LIN {X 0,Y 74.965,Z 475.117,A -85,B 0,C 180,E1 -28472.455,E2 -28472.455} C_VEL
LIN {X 0,Y 83.409,Z 481.852,A -85,B 0,C 180,E1 -28482.382,E2 -28482.382} C_VEL
LIN {X 0,Y 74.397,Z 477.881,A -85,B 0,C 180,E1 -28495.469,E2 -28495.469} C_VEL
LIN {X 0,Y 70.487,Z 473.263,A -85,B 0,C 180,E1 -28509.572,E2 -28509.572} C_VEL
LIN {X 0,Y 70.589,Z 468.61,A -85,B 0,C 180,E1 -28521.407,E2 -28521.407} C_VEL
LIN {X 0,Y 70.63,Z 467.022,A -85,B 0,C 180,E1 -28524.286,E2 -28524.286} C_VEL
LIN {X 0,Y 69.492,Z 461.707,A -85,B 0,C 180,E1 -28531.445,E2 -28531.445} C_VEL
LIN {X 0,Y 68.716,Z 454,A -85,B 0,C 180,E1 -28540.307,E2 -28540.307} C_VEL
LIN {X 0,Y 69.422,Z 443.261,A -85,B 0,C 180,E1 -28550.746,E2 -28550.746} C_VEL
LIN {X 0,Y 71.921,Z 431.623,A -85,B 0,C 180,E1 -28560.049,E2 -28560.049} C_VEL
LIN {X 0,Y 75.979,Z 417.83,A -85,B 0,C 180,E1 -28568.631,E2 -28568.631} C_VEL
LIN {X 0,Y 81.232,Z 402.293,A -85,B 0,C 180,E1 -28575.922,E2 -28575.922} C_VEL
LIN {X 0,Y 86.552,Z 386.58,A -85,B 0,C 180,E1 -28581.398,E2 -28581.398} C_VEL
LIN {X 0,Y 91.626,Z 370.778,A -85,B 0,C 180,E1 -28585.538,E2 -28585.538} C_VEL
LIN {X 0,Y 96.789,Z 352.875,A -85,B 0,C 180,E1 -28589.013,E2 -28589.013} C_VEL
LIN {X 0,Y 100.755,Z 336.389,A -85,B 0,C 180,E1 -28591.399,E2 -28591.399} C_VEL
LIN {X 0,Y 117.928,Z 249.676,A -85,B 0,C 180,E1 -28599.784,E2 -28599.784} C_VEL
LIN {X 0,Y 111.457,Z 229.955,A -85,B 0,C 180,E1 -28605.629,E2 -28605.629} C_VEL
LIN {X 0,Y 106.456,Z 215.128,A -85,B 0,C 180,E1 -28610.832,E2 -28610.832} C_VEL
LIN {X 0,Y 100.434,Z 201.5,A -85,B 0,C 180,E1 -28617.368,E2 -28617.368} C_VEL
LIN {X 0,Y 95.851,Z 191.545,A -85,B 0,C 180,E1 -28623.349,E2 -28623.349} C_VEL
LIN {X 0,Y 95.342,Z 190.433,A -85,B 0,C 180,E1 -28624.09,E2 -28624.09} C_VEL
LIN {X 0,Y 94.098,Z 188.156,A -85,B 0,C 180,E1 -28625.868,E2 -28625.868} C_VEL
LIN {X 0,Y 91.794,Z 185.771,A -85,B 0,C 180,E1 -28628.886,E2 -28628.886} C_VEL
LIN {X 0,Y 87.617,Z 183.57,A -85,B 0,C 180,E1 -28634.566,E2 -28634.566} C_VEL
LIN {X 0,Y 83.404,Z 181.257,A -85,B 0,C 180,E1 -28642.168,E2 -28642.168} C_VEL
LIN {X 0,Y 81.676,Z 178.087,A -85,B 0,C 180,E1 -28647.777,E2 -28647.777} C_VEL
LIN {X 0,Y 79.271,Z 173.794,A -85,B 0,C 180,E1 -28663.544,E2 -28663.544} C_VEL
LIN {X 0,Y 79.279,Z 173.506,A -85,B 0,C 180,E1 -28665.17,E2 -28665.17} C_VEL
LIN {X 0,Y 79.314,Z 173.871,A -85,B 0,C 180,E1 -28670.55,E2 -28670.55} C_VEL
LIN {X 0,Y 81.35,Z 177.859,A -85,B 0,C 180,E1 -28684.412,E2 -28684.412} C_VEL
LIN {X 0,Y 82.16,Z 178.643,A -85,B 0,C 180,E1 -28686.927,E2 -28686.927} C_VEL
LIN {X 0,Y 84.136,Z 181.84,A -85,B 0,C 180,E1 -28692.614,E2 -28692.614} C_VEL
LIN {X 0,Y 84.952,Z 183.183,A -85,B 0,C 180,E1 -28694.567,E2 -28694.567} C_VEL
LIN {X 0,Y 87.819,Z 187.557,A -85,B 0,C 180,E1 -28700.357,E2 -28700.357} C_VEL
LIN {X 0,Y 92.327,Z 197.444,A -85,B 0,C 180,E1 -28708.303,E2 -28708.303} C_VEL
LIN {X 0,Y 96.622,Z 207.533,A -85,B 0,C 180,E1 -28714.449,E2 -28714.449} C_VEL
LIN {X 0,Y 100.849,Z 217.771,A -85,B 0,C 180,E1 -28719.571,E2 -28719.571} C_VEL
LIN {X 0,Y 106.521,Z 232.316,A -85,B 0,C 180,E1 -28725.538,E2 -28725.538} C_VEL
LIN {X 0,Y 110.247,Z 242.256,A -85,B 0,C 180,E1 -28729.001,E2 -28729.001} C_VEL
LIN {X 0,Y 93.58,Z 323.333,A -85,B 0,C 180,E1 -28736.984,E2 -28736.984} C_VEL
LIN {X 0,Y 89.059,Z 341.545,A -85,B 0,C 180,E1 -28739.766,E2 -28739.766} C_VEL
LIN {X 0,Y 84.095,Z 358.706,A -85,B 0,C 180,E1 -28743.308,E2 -28743.308} C_VEL
LIN {X 0,Y 78.234,Z 376.248,A -85,B 0,C 180,E1 -28748.184,E2 -28748.184} C_VEL
LIN {X 0,Y 72.432,Z 392.761,A -85,B 0,C 180,E1 -28754.47,E2 -28754.47} C_VEL
LIN {X 0,Y 67.164,Z 407.561,A -85,B 0,C 180,E1 -28762.065,E2 -28762.065} C_VEL
LIN {X 0,Y 63.372,Z 419.467,A -85,B 0,C 180,E1 -28770.062,E2 -28770.062} C_VEL
LIN {X 0,Y 60.505,Z 430.86,A -85,B 0,C 180,E1 -28779.606,E2 -28779.606} C_VEL
LIN {X 0,Y 58.901,Z 442.203,A -85,B 0,C 180,E1 -28791.422,E2 -28791.422} C_VEL
LIN {X 0,Y 59.047,Z 450.62,A -85,B 0,C 180,E1 -28801.704,E2 -28801.704} C_VEL
LIN {X 0,Y 60.281,Z 457.783,A -85,B 0,C 180,E1 -28811.772,E2 -28811.772} C_VEL
LIN {X 0,Y 62.194,Z 463.073,A -85,B 0,C 180,E1 -28819.815,E2 -28819.815} C_VEL
LIN {X 0,Y 69.369,Z 472.869,A -85,B 0,C 180,E1 -28835.445,E2 -28835.445} C_VEL
LIN {X 0,Y 74.222,Z 476.893,A -85,B 0,C 180,E1 -28841.514,E2 -28841.514} C_VEL
LIN {X 0,Y 74.696,Z 477.491,A -85,B 0,C 180,E1 -28843.722,E2 -28843.722} C_VEL
LIN {X 0,Y 66.744,Z 473.028,A -85,B 0,C 180,E1 -28858.227,E2 -28858.227} C_VEL
LIN {X 0,Y 64.134,Z 467.784,A -85,B 0,C 180,E1 -28874.096,E2 -28874.096} C_VEL
LIN {X 0,Y 64.414,Z 465.191,A -85,B 0,C 180,E1 -28880.573,E2 -28880.573} C_VEL
LIN {X 0,Y 64.208,Z 463.497,A -85,B 0,C 180,E1 -28883.712,E2 -28883.712} C_VEL
LIN {X 0,Y 62.63,Z 456.544,A -85,B 0,C 180,E1 -28893.212,E2 -28893.212} C_VEL
LIN {X 0,Y 62.089,Z 448.132,A -85,B 0,C 180,E1 -28903.08,E2 -28903.08} C_VEL
LIN {X 0,Y 63.459,Z 436.622,A -85,B 0,C 180,E1 -28914.534,E2 -28914.534} C_VEL
LIN {X 0,Y 66.391,Z 425.073,A -85,B 0,C 180,E1 -28923.758,E2 -28923.758} C_VEL
LIN {X 0,Y 70.688,Z 411.53,A -85,B 0,C 180,E1 -28932.147,E2 -28932.147} C_VEL
LIN {X 0,Y 75.931,Z 396.902,A -85,B 0,C 180,E1 -28938.897,E2 -28938.897} C_VEL
LIN {X 0,Y 81.836,Z 379.941,A -85,B 0,C 180,E1 -28944.666,E2 -28944.666} C_VEL
LIN {X 0,Y 87.581,Z 362.016,A -85,B 0,C 180,E1 -28949.044,E2 -28949.044} C_VEL
LIN {X 0,Y 92.745,Z 343.45,A -85,B 0,C 180,E1 -28952.265,E2 -28952.265} C_VEL
LIN {X 0,Y 96.883,Z 324.277,A -85,B 0,C 180,E1 -28954.733,E2 -28954.733} C_VEL
LIN {X 0,Y 111.797,Z 251.982,A -85,B 0,C 180,E1 -28961.71,E2 -28961.71} C_VEL
LIN {X 0,Y 111.76,Z 250.857,A -85,B 0,C 180,E1 -28961.912,E2 -28961.912} C_VEL
LIN {X 0,Y 105.421,Z 230.727,A -85,B 0,C 180,E1 -28968.344,E2 -28968.344} C_VEL
LIN {X 0,Y 101.615,Z 219.129,A -85,B 0,C 180,E1 -28972.741,E2 -28972.741} C_VEL
LIN {X 0,Y 96.472,Z 206.764,A -85,B 0,C 180,E1 -28978.941,E2 -28978.941} C_VEL
LIN {X 0,Y 92.138,Z 196.752,A -85,B 0,C 180,E1 -28985.205,E2 -28985.205} C_VEL
LIN {X 0,Y 88.779,Z 189.564,A -85,B 0,C 180,E1 -28990.952,E2 -28990.952} C_VEL
LIN {X 0,Y 86.23,Z 185.464,A -85,B 0,C 180,E1 -28995.71,E2 -28995.71} C_VEL
LIN {X 0,Y 84.322,Z 182.251,A -85,B 0,C 180,E1 -29000.067,E2 -29000.067} C_VEL
LIN {X 0,Y 83.404,Z 181.257,A -85,B 0,C 180,E1 -29002.168,E2 -29002.168} C_VEL
LIN {X 0,Y 82.252,Z 180.805,A -85,B 0,C 180,E1 -29004.775,E2 -29004.775} C_VEL
LIN {X 0,Y 80.152,Z 181.741,A -85,B 0,C 180,E1 -29009.222,E2 -29009.222} C_VEL
LIN {X 0,Y 78.457,Z 182.828,A -85,B 0,C 180,E1 -29013.895,E2 -29013.895} C_VEL
LIN {X 0,Y 77.851,Z 182.595,A -85,B 0,C 180,E1 -29016.798,E2 -29016.798} C_VEL
LIN {X 0,Y 77.503,Z 180.426,A -85,B 0,C 180,E1 -29024.799,E2 -29024.799} C_VEL
LIN {X 0,Y 77.51,Z 180.763,A -85,B 0,C 180,E1 -29030.219,E2 -29030.219} C_VEL
LIN {X 0,Y 79.585,Z 184.776,A -85,B 0,C 180,E1 -29044.641,E2 -29044.641} C_VEL
LIN {X 0,Y 82.204,Z 189.209,A -85,B 0,C 180,E1 -29052.846,E2 -29052.846} C_VEL
LIN {X 0,Y 84.796,Z 193.632,A -85,B 0,C 180,E1 -29058.745,E2 -29058.745} C_VEL
LIN {X 0,Y 88.506,Z 202.301,A -85,B 0,C 180,E1 -29066.083,E2 -29066.083} C_VEL
LIN {X 0,Y 92.61,Z 212.637,A -85,B 0,C 180,E1 -29072.682,E2 -29072.682} C_VEL
LIN {X 0,Y 96.354,Z 222.347,A -85,B 0,C 180,E1 -29077.764,E2 -29077.764} C_VEL
LIN {X 0,Y 101.43,Z 235.842,A -85,B 0,C 180,E1 -29083.645,E2 -29083.645} C_VEL
LIN {X 0,Y 104.372,Z 244.207,A -85,B 0,C 180,E1 -29086.71,E2 -29086.71} C_VEL
LIN {X 0,Y 87.257,Z 324.229,A -85,B 0,C 180,E1 -29094.813,E2 -29094.813} C_VEL
LIN {X 0,Y 82.401,Z 342.673,A -85,B 0,C 180,E1 -29097.762,E2 -29097.762} C_VEL
LIN {X 0,Y 77.248,Z 359.578,A -85,B 0,C 180,E1 -29101.467,E2 -29101.467} C_VEL
LIN {X 0,Y 71.316,Z 376.654,A -85,B 0,C 180,E1 -29106.537,E2 -29106.537} C_VEL
LIN {X 0,Y 65.229,Z 393.074,A -85,B 0,C 180,E1 -29113.342,E2 -29113.342} C_VEL
LIN {X 0,Y 59.393,Z 409.18,A -85,B 0,C 180,E1 -29122.667,E2 -29122.667} C_VEL
LIN {X 0,Y 55.028,Z 423.179,A -85,B 0,C 180,E1 -29133.855,E2 -29133.855} C_VEL
LIN {X 0,Y 52.601,Z 435.247,A -85,B 0,C 180,E1 -29146.477,E2 -29146.477} C_VEL
LIN {X 0,Y 52.302,Z 445.883,A -85,B 0,C 180,E1 -29159.999,E2 -29159.999} C_VEL
LIN {X 0,Y 53.572,Z 453.604,A -85,B 0,C 180,E1 -29171.348,E2 -29171.348} C_VEL
LIN {X 0,Y 56.584,Z 461.251,A -85,B 0,C 180,E1 -29183.807,E2 -29183.807} C_VEL
LIN {X 0,Y 65.15,Z 471.324,A -85,B 0,C 180,E1 -29200.333,E2 -29200.333} C_VEL
LIN {X 0,Y 67.679,Z 473.354,A -85,B 0,C 180,E1 -29203.367,E2 -29203.367} C_VEL
LIN {X 0,Y 60.346,Z 468.762,A -85,B 0,C 180,E1 -29218.388,E2 -29218.388} C_VEL
LIN {X 0,Y 58.169,Z 463.057,A -85,B 0,C 180,E1 -29236.012,E2 -29236.012} C_VEL
LIN {X 0,Y 58.19,Z 461.195,A -85,B 0,C 180,E1 -29240.46,E2 -29240.46} C_VEL
LIN {X 0,Y 57.189,Z 457.794,A -85,B 0,C 180,E1 -29245.925,E2 -29245.925} C_VEL
LIN {X 0,Y 55.658,Z 449.518,A -85,B 0,C 180,E1 -29257.249,E2 -29257.249} C_VEL
LIN {X 0,Y 55.981,Z 438.551,A -85,B 0,C 180,E1 -29270.191,E2 -29270.191} C_VEL
LIN {X 0,Y 58.93,Z 425.433,A -85,B 0,C 180,E1 -29282.542,E2 -29282.542} C_VEL
LIN {X 0,Y 63.534,Z 411.067,A -85,B 0,C 180,E1 -29292.645,E2 -29292.645} C_VEL
LIN {X 0,Y 69.352,Z 395.353,A -85,B 0,C 180,E1 -29300.591,E2 -29300.591} C_VEL
LIN {X 0,Y 75.139,Z 379.462,A -85,B 0,C 180,E1 -29306.37,E2 -29306.37} C_VEL
LIN {X 0,Y 80.933,Z 362.059,A -85,B 0,C 180,E1 -29310.896,E2 -29310.896} C_VEL
LIN {X 0,Y 86.256,Z 343.945,A -85,B 0,C 180,E1 -29314.23,E2 -29314.23} C_VEL
LIN {X 0,Y 90.647,Z 324.616,A -85,B 0,C 180,E1 -29316.857,E2 -29316.857} C_VEL
LIN {X 0,Y 105.846,Z 253.711,A -85,B 0,C 180,E1 -29323.88,E2 -29323.88} C_VEL
LIN {X 0,Y 105.757,Z 252.112,A -85,B 0,C 180,E1 -29324.205,E2 -29324.205} C_VEL
LIN {X 0,Y 99.794,Z 232.307,A -85,B 0,C 180,E1 -29331.025,E2 -29331.025} C_VEL
LIN {X 0,Y 96.721,Z 222.592,A -85,B 0,C 180,E1 -29335.036,E2 -29335.036} C_VEL
LIN {X 0,Y 92.072,Z 210.898,A -85,B 0,C 180,E1 -29341.318,E2 -29341.318} C_VEL
LIN {X 0,Y 88.434,Z 201.843,A -85,B 0,C 180,E1 -29347.278,E2 -29347.278} C_VEL
LIN {X 0,Y 85.491,Z 195.177,A -85,B 0,C 180,E1 -29352.937,E2 -29352.937} C_VEL
LIN {X 0,Y 83.411,Z 191.521,A -85,B 0,C 180,E1 -29357.319,E2 -29357.319} C_VEL
LIN {X 0,Y 81.76,Z 188.617,A -85,B 0,C 180,E1 -29361.45,E2 -29361.45} C_VEL
LIN {X 0,Y 79.687,Z 185.01,A -85,B 0,C 180,E1 -29368.128,E2 -29368.128} C_VEL
LIN {X 0,Y 77.851,Z 182.595,A -85,B 0,C 180,E1 -29376.798,E2 -29376.798} C_VEL
LIN {X 0,Y 77.437,Z 182.463,A -85,B 0,C 180,E1 -29379.671,E2 -29379.671} C_VEL
LIN {X 0,Y 76.717,Z 183.728,A -85,B 0,C 180,E1 -29383.455,E2 -29383.455} C_VEL
LIN {X 0,Y 75.711,Z 188.287,A -85,B 0,C 180,E1 -29392.078,E2 -29392.078} C_VEL
LIN {X 0,Y 77.695,Z 191.936,A -85,B 0,C 180,E1 -29404.765,E2 -29404.765} C_VEL
LIN {X 0,Y 79.629,Z 195.522,A -85,B 0,C 180,E1 -29411.349,E2 -29411.349} C_VEL
LIN {X 0,Y 81.77,Z 199.47,A -85,B 0,C 180,E1 -29416.811,E2 -29416.811} C_VEL
LIN {X 0,Y 84.893,Z 207.401,A -85,B 0,C 180,E1 -29423.862,E2 -29423.862} C_VEL
LIN {X 0,Y 88.583,Z 217.478,A -85,B 0,C 180,E1 -29430.627,E2 -29430.627} C_VEL
LIN {X 0,Y 92.663,Z 228.696,A -85,B 0,C 180,E1 -29436.743,E2 -29436.743} C_VEL
LIN {X 0,Y 97.908,Z 243.895,A -85,B 0,C 180,E1 -29443.377,E2 -29443.377} C_VEL
LIN {X 0,Y 98.644,Z 246.058,A -85,B 0,C 180,E1 -29444.221,E2 -29444.221} C_VEL
LIN {X 0,Y 81.174,Z 324.439,A -85,B 0,C 180,E1 -29452.283,E2 -29452.283} C_VEL
LIN {X 0,Y 75.882,Z 343.629,A -85,B 0,C 180,E1 -29455.44,E2 -29455.44} C_VEL
LIN {X 0,Y 70.406,Z 360.643,A -85,B 0,C 180,E1 -29459.404,E2 -29459.404} C_VEL
LIN {X 0,Y 63.567,Z 379.158,A -85,B 0,C 180,E1 -29465.471,E2 -29465.471} C_VEL
LIN {X 0,Y 57.508,Z 394.806,A -85,B 0,C 180,E1 -29472.839,E2 -29472.839} C_VEL
LIN {X 0,Y 51.637,Z 410.584,A -85,B 0,C 180,E1 -29483.454,E2 -29483.454} C_VEL
LIN {X 0,Y 47.544,Z 423.904,A -85,B 0,C 180,E1 -29496.013,E2 -29496.013} C_VEL
LIN {X 0,Y 45.715,Z 434.463,A -85,B 0,C 180,E1 -29508.92,E2 -29508.92} C_VEL
LIN {X 0,Y 45.993,Z 445.115,A -85,B 0,C 180,E1 -29524.381,E2 -29524.381} C_VEL
LIN {X 0,Y 47.97,Z 452.754,A -85,B 0,C 180,E1 -29537.038,E2 -29537.038} C_VEL
LIN {X 0,Y 51.337,Z 459.312,A -85,B 0,C 180,E1 -29548.629,E2 -29548.629} C_VEL
LIN {X 0,Y 58.141,Z 466.908,A -85,B 0,C 180,E1 -29561.615,E2 -29561.615} C_VEL
LIN {X 0,Y 59.58,Z 468.276,A -85,B 0,C 180,E1 -29564.941,E2 -29564.941} C_VEL
LIN {X 0,Y 53.279,Z 463.124,A -85,B 0,C 180,E1 -29582.499,E2 -29582.499} C_VEL
LIN {X 0,Y 52.267,Z 459.406,A -85,B 0,C 180,E1 -29594.394,E2 -29594.394} C_VEL
LIN {X 0,Y 52.185,Z 457.906,A -85,B 0,C 180,E1 -29598.34,E2 -29598.34} C_VEL
LIN {X 0,Y 50.575,Z 453.266,A -85,B 0,C 180,E1 -29606.011,E2 -29606.011} C_VEL
LIN {X 0,Y 49.018,Z 444.929,A -85,B 0,C 180,E1 -29618.238,E2 -29618.238} C_VEL
LIN {X 0,Y 49.763,Z 433.322,A -85,B 0,C 180,E1 -29632.848,E2 -29632.848} C_VEL
LIN {X 0,Y 52.936,Z 420.701,A -85,B 0,C 180,E1 -29645.41,E2 -29645.41} C_VEL
LIN {X 0,Y 58.278,Z 405.539,A -85,B 0,C 180,E1 -29656.343,E2 -29656.343} C_VEL
LIN {X 0,Y 64.076,Z 390.489,A -85,B 0,C 180,E1 -29663.982,E2 -29663.982} C_VEL
LIN {X 0,Y 70.062,Z 374.392,A -85,B 0,C 180,E1 -29669.732,E2 -29669.732} C_VEL
LIN {X 0,Y 76.113,Z 356.627,A -85,B 0,C 180,E1 -29674.186,E2 -29674.186} C_VEL
LIN {X 0,Y 81.364,Z 338.54,A -85,B 0,C 180,E1 -29677.383,E2 -29677.383} C_VEL
LIN {X 0,Y 87.325,Z 311.516,A -85,B 0,C 180,E1 -29680.81,E2 -29680.81} C_VEL
LIN {X 0,Y 100.062,Z 255.064,A -85,B 0,C 180,E1 -29686.305,E2 -29686.305} C_VEL
LIN {X 0,Y 99.799,Z 253.33,A -85,B 0,C 180,E1 -29686.769,E2 -29686.769} C_VEL
LIN {X 0,Y 94.554,Z 234.798,A -85,B 0,C 180,E1 -29693.628,E2 -29693.628} C_VEL
LIN {X 0,Y 92.123,Z 226.64,A -85,B 0,C 180,E1 -29697.236,E2 -29697.236} C_VEL
LIN {X 0,Y 87.859,Z 215.139,A -85,B 0,C 180,E1 -29703.809,E2 -29703.809} C_VEL
LIN {X 0,Y 84.605,Z 206.38,A -85,B 0,C 180,E1 -29709.948,E2 -29709.948} C_VEL
LIN {X 0,Y 82.38,Z 200.914,A -85,B 0,C 180,E1 -29714.83,E2 -29714.83} C_VEL
LIN {X 0,Y 79.926,Z 196.3,A -85,B 0,C 180,E1 -29720.855,E2 -29720.855} C_VEL
LIN {X 0,Y 79.125,Z 194.81,A -85,B 0,C 180,E1 -29723.23,E2 -29723.23} C_VEL
LIN {X 0,Y 77.311,Z 191.353,A -85,B 0,C 180,E1 -29729.99,E2 -29729.99} C_VEL
LIN {X 0,Y 75.677,Z 187.448,A -85,B 0,C 180,E1 -29744.77,E2 -29744.77} C_VEL
LIN {X 0,Y 75.704,Z 187.458,A -85,B 0,C 180,E1 -29749.071,E2 -29749.071} C_VEL
LIN {X 0,Y 75.711,Z 188.287,A -85,B 0,C 180,E1 -29752.078,E2 -29752.078} C_VEL
LIN {X 0,Y 75.79,Z 190.401,A -85,B 0,C 180,E1 -29756.269,E2 -29756.269} C_VEL
LIN {X 0,Y 76.088,Z 195.438,A -85,B 0,C 180,E1 -29762.727,E2 -29762.727} C_VEL
LIN {X 0,Y 76.718,Z 199.909,A -85,B 0,C 180,E1 -29767.72,E2 -29767.72} C_VEL
LIN {X 0,Y 78.057,Z 203.875,A -85,B 0,C 180,E1 -29772.788,E2 -29772.788} C_VEL
LIN {X 0,Y 78.98,Z 205.843,A -85,B 0,C 180,E1 -29775.327,E2 -29775.327} C_VEL
